// ---- GlobalTextList.TcGTLO
TEXTLIST GlobalTextList
  4330 = '\tPCW behavior Condition  (Suggestion from Intel)\n\tPCW SUPPLY THERMOCOUPLE LH\xa0 > 14°C, Warning: “PCW supply high temp”, Action: Nil\n\t(Tester) Incoming pressure for 6bar LH <550 kPa , Warning: “6 bar OFA LH air pressure low”,\xa0 Action: Nil\n\t(AP) Incoming pressure for 9 bar\xa0 LH < 850kPa, Warning:\xa0 “9 bar OFA LH air pressure low”, Action: Nil\n\tPCW Return Temperature – PCW Supply Temperature > 10degC, Warning: “Excessive heat load into PCW”, Action = Nil\n\tT-BOT Dew Point - PCW Supply Temperature > -2degC, Warning : “Dew point – PCW temperature above control limit, condensation warning.”, Action = Nil\n\tT-BOT Dew Point - PCW Supply Temperature > 0degC, Alarm: “Dew point – PCW temperature above critical control limit, condensation alarm.”, Action = Shut off PCW Supply and Return\n\tIf Either One of the Leak Sensor is Trigger, Alarm: “System PCW Leakage .”, Action = Shut off PCW Supply and Return.\n\t'
  1821 = '\tPCW behavior Condition  (Suggestion from Intel)\n\tPCW SUPPLY THERMOCOUPLE \xa0 > 14°C, Warning: “PCW supply high temp”, Action: Nil\n\t(Tester) Incoming pressure for 6bar  <550 kPa , Warning: “6 bar OFA LH air pressure low”,\xa0 Action: Nil\n\t(AP) Incoming pressure for 9 bar\xa0    < 850kPa, Warning:\xa0 “9 bar OFA LH air pressure low”, Action: Nil\n\tPCW Return Temperature – PCW Supply Temperature > 10degC, Warning: “Excessive heat load into PCW”, Action = Nil\n\tDew Point - PCW Supply Temperature > -2degC, Warning : “Dew point – PCW temperature above control limit, condensation warning.”, Action = Nil\n\tDew Point - PCW Supply Temperature > 0degC, Alarm: “Dew point – PCW temperature above critical control limit, condensation alarm.”, Action = Shut off PCW Supply and Return\n\tIf Either One of the Leak Sensor is Trigger, Alarm: “System PCW Leakage .”, Action = Shut off PCW Supply and Return.\n\t'
  3264 = '\tPCW behavior Condition  (Suggestion from Intel)\n\tPCW SUPPLY THERMOCOUPLE \xa0 > 14°C, Warning: “PCW supply high temp”, Action: Nil\n\t(Tester) Incoming pressure for 6bar  <550 kPa , Warning: “6 bar OFA LH air pressure low”,\xa0 Action: Nil\n\t(AP) Incoming pressure for 9 bar\xa0    < 850kPa, Warning:\xa0 “9 bar OFA LH air pressure low”, Action: Nil\n\tPCW Return Temperature – PCW Supply Temperature > 10degC, Warning: “Excessive heat load into PCW”, Action = Nil\n\tT-BOT Dew Point - PCW Supply Temperature > -2degC, Warning : “Dew point – PCW temperature above control limit, condensation warning.”, Action = Nil\n\tT-BOT Dew Point - PCW Supply Temperature > 0degC, Alarm: “Dew point – PCW temperature above critical control limit, condensation alarm.”, Action = Shut off PCW Supply and Return\n\tIf Either One of the Leak Sensor is Trigger, Alarm: “System PCW Leakage .”, Action = Shut off PCW Supply and Return.\n\t'
  571 = ' : '
  2622 = ' : AP Power Signal is not detected    '
  2268 = ' : AP Present Signal is not detected  '
  613 = ' : AP Ready Signal is not detected  '
  2271 = ' : APDeactuatedHwr Signal is not detected   '
  2182 = ' : APDeactuatedPLC Signal is not detected '
  2896 = ' : Cell Door Closed  Signal is not detected'
  3152 = ' : Cell Door Locked Signal is not detected'
  1060 = ' : Cell Fluid Leakage1 Signal is detected   '
  1608 = ' : Cell Fluid Leakage2  Signal is detecte'
  881 = ' : Cell Ground Fault Signal is detected     '
  4213 = ' : Debug Station Facility Ac Power OFF'
  3618 = ' : Debug Station Facility Ac Power OFF Detected'
  4041 = ' : DS cell fluid leakage 1 Signal is Detected'
  3638 = ' : DS cell fluid leakage 2 signal is detected'
  5457 = ' : e6BarLowOFAAirPressureAlarm'
  634 = ' : e6BarLowOFAAirPressureWarning'
  2402 = ' : e9BarLowOFAAirPressureWarning '
  3302 = ' : eCondensationWarning'
  639 = ' : eCriticalCondensationAlarm'
  244 = ' : eExcessiveHeatLoadIntoPCWWarning  '
  2432 = ' : ePCWSupplyHighTempWarning'
  6407 = ' : eSystemPCWLeakage2Alarm'
  1774 = ' : eSystemPCWLeakageAlarm'
  959 = ' : eSystemPCWReturnLeakageAlarm'
  3498 = ' : eSystemPCWSupplyLeakageAlarm'
  1221 = ' : Front Side Door Lock Signal is not Detected'
  3416 = ' : ipTCDrawerCylDown signal not detected'
  3147 = ' : ipTCDrawerCylExtendRS Signal not detected'
  1457 = ' : ipTCDrawerCylExtendRS signal not detected'
  3399 = ' : ipTCDrawerCylExtendRSError'
  1978 = ' : ipTCDrawerCylRetractRS signal not detected'
  7 = ' : ipTCDrawerCylRetractRSError'
  2361 = ' : ipTCDrawerCylUp signal not detected'
  137 = ' : nnnnn'
  1011 = ' : TBOT ANTI-COLLISION TRIGGERED SIGNAL'
  4581 = ' : TBot EAP AC Power OFF Detected'
  618 = ' : TBotEAPACPowerOFFDetected'
  2835 = ' : Tester Latches Closed  Signal is not detected '
  3173 = ' : Tester Present Signal is not detected  '
  2325 = ' : Tester Ready Signal is not detected  '
  700 = ' : TesterPower On  Signal is not detected '
  1694 = ' : TIU DOWN SOLENOID'
  957 = ' : TIU DOWN Solenoid Valve'
  4475 = ' : TIU EXTEND REED SWITCH'
  3125 = ' : TIU EXTEND SOLENOID'
  1932 = ' : TIU EXTEND Solenoid Valve'
  3331 = ' : TIU NOT SAFE TO MOVE'
  2540 = ' : TIU NOT SAFE TO MOVE (True: Not Safe, False Safe)'
  3756 = ' : TIU NOT SAFE TO MOVE (True:Not Safe,False: Safe)'
  3605 = ' : TIU NOT SAFETOMOVE (True:Not Safe,False: Safe)'
  1787 = ' : TIU Present Signal is not detected   '
  1466 = ' : TIU RETRACT REED SWITCH'
  1952 = ' : TIU RETRACT SOLENOID'
  2863 = ' : TIU RETRACT Solenoid Valve'
  4 = ' : TIU UP SOLENOID'
  1350 = ' : TIU UP Solenoid Valve'
  1123 = ' :(----------------------------------------------------------)'
  630 = ' :(--------------------------------------------------------------)'
  1673 = ' :(--------------------------------------------------------------------------------)'
  98 = ' :AP is not in UP Position'
  369 = ' :Both TIU Extern & Retract  Signal  are Detected'
  644 = ' :Both TIU Up & Down  Signal  are Detected'
  752 = ' :Door Close Signal is not Detected'
  2348 = ' :Door Lock Signal is not Detected'
  895 = ' :DrawerDownError'
  1112 = ' :DrawerExtendError'
  2406 = ' :DrawerRetractError'
  1818 = ' :DrawerUpError'
  4103 = ' :ipTCDrawerCylExtendRSError'
  1922 = ' :TBot EAP AntiCollision Triggered'
  4187 = ' :TBot EAP Not Safe To Move Error'
  2535 = ' :TBot EAPNotSofeToMoveError'
  2562 = ' :TBot Side Door Close Signal is not Detected'
  1220 = ' :TBot Side Door Lock Signal is not Detected'
  1668 = ' :TCC Session Active'
  4906 = '%3f'
  6313 = '%4.2'
  6022 = '%4.2f'
  1391 = '%5.0f'
  6312 = '%5.2'
  1806 = '%5.2f'
  2996 = '%6.3f'
  313 = '%d'
  5400 = '%D'
  311 = '%f'
  991 = '%i'
  4616 = '%s'
  3443 = '%t'
  3829 = "'C"
  1185 = '(----------------------------------------------------------------------------------)'
  632 = '(AP) OFA 10 bar Leak Flow'
  1515 = '(AP) OFA Pressure 10 bar'
  22 = '(Tester) OFA 6 bar Leak Flow'
  3541 = '(Tester) OFA Pressure 6 bar'
  4601 = '---------'
  234 = '01)Column Leakage'
  826 = '01)Col_Leakage'
  710 = '01)_AP_PresentSensor'
  3291 = '01)_AP_PresentSensor*'
  322 = '01)_Column Leakage'
  151 = '01)_ColumnLeakage'
  393 = '01)_Col_Leakage'
  427 = '02)_AllDrawerRetractedInCell'
  348 = '02)_All_Dwr_Ret'
  683 = '02)_AP_PowerOn'
  5106 = '02)_AP_PowerOn*'
  303 = '03)ColumnGround'
  976 = '03)_AP_Ready'
  75 = '03)_ColumnGround'
  941 = '03)_Col_Grd_Falt'
  1133 = '03)_Col_Grund_Falt'
  43 = '04)_AP_DeactuatedPLC'
  1100 = '04)_AP_DeactuatedPLC`*`'
  785 = '05)_AP_DeactuatedHwr'
  5223 = '05)_AP_DeactuatedHwr`*`'
  977 = '06)_CellFluidLeakage1'
  988 = '07)_CellFluidLeakage2'
  877 = '08)_CellGroundFault'
  421 = '09)_TesterPresent'
  2063 = '09)_TesterPresent*'
  2493 = '09)_TesterPresent**'
  1062 = '1'
  460 = "1'AP_PresentSenser"
  321 = '1)  AP_PresentSenser'
  671 = '1) AP_PresentSenser'
  566 = '1)_AP_PresentSensor'
  745 = '1)_Col_Leakage'
  537 = '1-AP_PresentSenser'
  2484 = '1. opDBStnMainPCWSupply'
  433 = '10)_TesterPowerOn'
  607 = '10)_TesterPowerOn*'
  729 = '10)_TesterPowerOn**'
  131 = '11)_TesterReady   '
  621 = '12)_TCCellDoorClosed\t'
  278 = '13)_TesterLatchesClosed'
  920 = '13)_TesterLatchesClosed**'
  117 = '14)_TIUPresent\t'
  577 = '2) AP_PowerOn'
  756 = '2)AP_PowerOn'
  129 = '2)_All_Dwr_Ret'
  628 = '2)_AP_PowerOn'
  1565 = '2. opDBStnPCWSupplyPurge'
  1692 = '21'
  2299 = '240 Power and PCW'
  4252 = '240v AP Power'
  5206 = '240v AP Power Feedback'
  2620 = '240v AP Power Feedback (Input)'
  4573 = '240v AP Power Feedback(Input)'
  2171 = '240v AP Power(Output)'
  4256 = '240v DPS/Tester Power'
  3856 = '240v Tester Power Feedback(Input)'
  1480 = '240v Tester Power(Output)'
  2285 = '240vTester Power(Output)'
  3074 = '240vTesterPower(Output)'
  846 = '3) AP_Ready'
  370 = '3)AP_Ready'
  145 = '3)_AP_Ready'
  1595 = '3)_Col_Grd'
  705 = '3)_Col_Grd_Falt'
  6218 = '3. opDBStnMainPCWReturn'
  84 = '4) AP_DeactuatedPLC'
  534 = '4)AP_DeactuatedPLC'
  965 = '4)_AP_DeactuatedPLC'
  1662 = '4. opDBStnPCWAWN'
  503 = '5) AP_DeactuatedHwr'
  559 = '5)AP_DeactuatedHwr'
  85 = '5)_AP_DeactuatedHwr'
  6470 = '5. opDBStnSupplyAirPurge'
  104 = '6)_CellFluidLeakage1'
  2776 = '6. opDBStnLeakFlowPCWValve'
  144 = '7)_CellFluidLeakage2'
  2027 = '7. opDBStnLowFlowPCWValve'
  51 = '8)_CellGroundFault'
  139 = '9)_TesterPresent'
  1420 = ': ColumnAlarmBit1'
  175 = ': ColumnAlarmBit2'
  658 = ': ColumnAlarmBit3'
  2042 = ': e6BarLowOFAAirPressureAlarm'
  5458 = ': ipTCDrawerCylRetractRSError'
  3543 = ': TBOT ANTI-COLLISION TRIGGERED SIGNAL'
  2700 = ': TBOT ANTI-COLLISION TRIGGERED SOGNAL'
  2570 = ': TIU EXTEND REED SWITCH'
  2097 = ': TIU NOT SAFE TO MOVE'
  3354 = ': TIU RETRACT REED SWITCH'
  2180 = ':AP is not in UP Position'
  4324 = ':ipTCDrawerCylRetractRSError'
  1467 = 'A'
  950 = 'AAAAAAAAAAA'
  3702 = 'Abort'
  2141 = 'Abort Running Timer'
  4237 = 'Abort Timer'
  5258 = 'Abort Timer (delay time)'
  312 = 'Actual Position'
  72 = 'Advanced'
  3639 = 'AH Alarm'
  3595 = 'AH Enable'
  4624 = 'AH SP'
  3633 = 'AHH Alarm'
  3579 = 'AHH Enable'
  3584 = 'AHH SP'
  2847 = 'Air Pressure Low'
  343 = 'Air Pressure Low ()'
  4556 = 'Air Pressure Low (Pressure is Less Than 550kpa)'
  2694 = 'Air Pressure Low (Pressure is less than 550kpa)'
  1084 = 'Air Pressure Low (Pressure is less than 850kPa)'
  3644 = 'AL Alarm'
  3600 = 'AL Enable'
  4631 = 'AL SP'
  5380 = 'Alar Auto Clearm'
  265 = 'Alarm'
  1301 = 'Alarm (Auto Clear)'
  1858 = 'Alarm Auto Clear'
  2577 = 'ALARM ID BIT STATUS'
  186 = 'ALARM ID BITS'
  690 = 'Alarm Reset'
  1223 = 'Alarm Running Timer'
  2152 = 'Alarm RunningTimer'
  2258 = 'Alarm Set PointWarning SetPoint'
  1212 = 'Alarm SetPoint'
  3433 = 'Alarm Timer'
  1638 = 'Alarm Timer (Second)'
  301 = 'Alarn Reset'
  3650 = 'ALL Alarm'
  3606 = 'ALL Enable'
  4638 = 'ALL SP'
  4995 = 'AllTCDrawer is not inside Cell'
  504 = 'AllTCDrawer_Not_In_Cell'
  5491 = 'AP 240Pwr Check Delay'
  1613 = 'AP Heater'
  1652 = 'AP HEATER_CURRENT'
  276 = 'AP is not in UP Position'
  5071 = 'AP Safe to Engage'
  2704 = 'AP240PwrCheck Delay(ms)'
  191 = 'AP240PwrCheckDelay(ms)'
  3283 = 'APReadyCheckDelay(ms)'
  81 = 'Auto'
  76 = 'Auto Input'
  624 = 'Auto Mode'
  469 = 'AutoRsetEvntTrigger'
  867 = 'BackDoorSimulationMode'
  1657 = 'Bar'
  633 = 'bar'
  252 = 'BH_HEATER_CURRENT_1'
  255 = 'BH_HEATER_CURRENT_2'
  254 = 'BH_HEATER_CURRENT_3'
  256 = 'BH_HEATER_CURRENT_4'
  1414 = 'BH_RTD_1'
  249 = 'BH_RTD_2'
  5795 = 'Btn No'
  1042 = 'Btn VIO Sim Override'
  6219 = 'Button'
  787 = 'Button: '
  1293 = 'ButtonModeConditionSimulation'
  1188 = 'ButtonModeConditionSimulation[iHMICbLevelSelection,iHMIBtnType]'
  535 = 'ButtonModeConditionSimulation[iHMICbLevelSelection,]'
  2089 = 'Cell Outputs :'
  1379 = 'Cell PCW'
  4038 = 'Cell Stack'
  2301 = 'CELL STACK'
  199 = 'Checkbox'
  2185 = 'Co'
  5100 = 'Col GroundFault'
  353 = 'COLUMN'
  2401 = 'Column'
  2816 = 'Column (AP) OFA Pressure 10 bar'
  329 = 'Column (Tester) OFA Pressure 6 bar'
  1708 = 'COLUMN ALARM ID BIT STATUS'
  4257 = 'COLUMN ALARM STATUS'
  2378 = 'Column Dew Point Sensor'
  3243 = 'Column Diagnostic Status'
  913 = 'Column Inputs :'
  90 = 'Column IO Diagnostic Mode'
  731 = 'Column Outputs :'
  2914 = 'Column PCW Leakage'
  3578 = 'Column PCW Regular Flow'
  2013 = 'Column PCW Return Pressure'
  2795 = 'Column PCW Return Temperature'
  2397 = 'Column PCW Supply Pressure'
  4011 = 'Column PCW Supply Temperature'
  1568 = 'Column Temperature'
  5977 = 'ColumnPCWLeakage2EAP'
  4652 = 'ColumnPCWLeakageEAP'
  2796 = 'ColumnPCWReturnLeakageEAP'
  760 = 'ColumnPCWSupplyLeakageEAP'
  5227 = 'Column_PCWLeakage'
  983 = 'Col_GroundFault'
  733 = 'Commands:'
  70 = 'Control'
  3437 = 'Current Value'
  272 = 'Cycle Running'
  4645 = 'DB'
  4543 = 'DBColumnPCWLeakage2EAP'
  3649 = 'DBColumnPCWLeakageEAP'
  4640 = 'DBColumnPCWReturnLeakageEAP'
  2584 = 'DBColumnPCWSupplyLeakageEAP'
  101 = 'DBColumnShutOffACPowerEAP'
  3120 = 'Dbug Station PCW Low Flow'
  270 = 'De Air Valve'
  1451 = 'De Pressure (Psi):'
  1001 = 'De Pressure Preset (Psi):'
  1464 = 'De Pressure Sen (Psi):'
  1689 = 'DE Stepping'
  4420 = 'DEBUG COLUMN ALARM ID BIT STATUS'
  3964 = 'DEBUG COLUMN ALARM STATUS'
  3330 = 'Debug Column Diagnostic Status'
  91 = 'Debug Column EAP Signals :'
  1164 = 'Debug Station'
  5185 = 'DEBUG STATION'
  2775 = 'Debug Station (AP) OFA 10 bar Leak Flow'
  1849 = 'Debug Station (Tester) OFA 6 bar Leak Flow'
  1416 = 'Debug Station Diagnostic Status'
  2458 = 'DEBUG STATION INPUTS'
  889 = 'DEBUG STATION IPC INPUTS'
  3105 = 'DEBUG STATION IPC OUTPUT'
  1865 = 'DEBUG STATION OUTPUT'
  271 = 'Debug Station PCW Leak Flow'
  488 = 'DeReg Pressure (Psi):'
  373 = 'DESolValve'
  541 = 'Development Purpose only'
  2911 = 'Dew Point '
  1678 = 'Dew Point - PCW Supply Temperature > -2degC, Warning :\nDew point – PCW temperature is above control limit, condensation warning'
  3845 = 'Dew Point - PCW Supply Temperature > -2degC, Warning : “Dew point – PCW temperature above control limit, condensation warning.”, Action = Nil'
  2334 = 'Dew Point - PCW Supply Temperature > 0degC, \nDew point – PCW temperature above critical control limit, condensation alarm\n'
  2414 = 'Dew Point - PCW Supply Temperature > 0degC, Alarm:\nDew point – PCW temperature above critical control limit, condensation alarm\n'
  4897 = 'Dew Point Alarm'
  3419 = 'Dew Point Dew Point '
  3035 = 'Dew Point Temperature'
  2356 = 'Dew Point Warning'
  1545 = 'Done Requested Action'
  1472 = 'Drawer In Request'
  1251 = 'Drawer Out Request'
  562 = 'Drawer Teaching Mode'
  1994 = 'DS_Facility_eapShutOffAllACPower'
  2386 = 'e6BarLowOFAAirPressureAlarm'
  398 = 'EAP SAFTY SIGNAL STATUS'
  1205 = 'EAP SAFTY SIGNAL STATUSSTATUS'
  2987 = 'EAP SIGNAL STATUS'
  3895 = 'eapShutOffAllACPower'
  948 = 'Enable'
  2173 = 'Enable Man: Stepping'
  1387 = 'Enable Man:Stepping'
  823 = 'Enable Manual Stepping Option'
  1120 = 'Enable Simulation'
  3674 = 'Enable/ Disable Status'
  1317 = 'EndPressure'
  2517 = 'EPT : '
  3022 = 'EPT States'
  314 = 'Error Code'
  4201 = 'Error Status: [ 0: No Error ]'
  1271 = 'Error Status: [0: No Error'
  2810 = 'ew Point Dew Point '
  83 = 'Extend'
  88 = 'Extended'
  2945 = 'F'
  2527 = 'Facility Alarm (Dew point & OFA6Bar)'
  3229 = 'Facility Alarm (Dew point & OFA6Bar) '
  4331 = 'Facility Alarm Set Default Timer and Point Value(Dew point & OFA6Bar) '
  4547 = 'Facility Alarm Set point and Timer'
  78 = 'Failed'
  80 = 'Failed to extend'
  79 = 'Failed to retract'
  1675 = 'For  Development And '
  4075 = 'Green: Enable , Gray: Disable'
  448 = 'Green:Enable , Gray: Disable'
  873 = 'GroupBox'
  3617 = 'Healthy'
  771 = 'Heater'
  1455 = 'HEATER_CURRENT_1'
  703 = 'HEATER_CURRENT_1:'
  1958 = 'HEATER_CURRENT_2'
  1131 = 'HEATER_CURRENT_3'
  500 = 'HEATER_CURRENT_4'
  1357 = 'Individual Alarm ID'
  1274 = 'Individual Alarm ID:'
  759 = 'Init All Level'
  3193 = 'INPUT'
  263 = 'Inputs :'
  636 = 'IO Diagnostic Mode'
  218 = 'ipAllTCDrawerRetractedinCell'
  734 = 'ipAPDeactuatedHwr'
  56 = 'ipAPDeactuatedPLC'
  715 = 'ipAPPowerOn'
  297 = 'ipAPPresentSensor'
  1003 = 'ipAPReady'
  409 = 'ipCellFluidLeakage1'
  994 = 'ipCellFluidLeakage2'
  611 = 'ipCellGroundFault'
  1030 = 'ipColumnFluid_PCW_Leakage'
  3804 = 'ipDBColumnPCWLeakage'
  1434 = 'ipDBColumnPCWLeakage2'
  777 = 'ipDBColumnPCWLeakageEAP'
  2983 = 'ipDBColumnPCWReturnLeakage'
  1794 = 'ipDBColumnPCWReturnLeakageEAP'
  631 = 'ipDBColumnPCWSupplyLeakage'
  3362 = 'ipDBColumnPCWSupplyLeakageEAP'
  2784 = 'ipDBStnAPDeactuatedHwr'
  1899 = 'ipDBStnAPDeactuatedPLC'
  1677 = 'ipDBStnAPPowerOn'
  1898 = 'ipDBStnAPPresentSensor'
  1372 = 'ipDBStnAPReady'
  2044 = 'ipDBStnCellFluidLeakage1'
  4211 = 'ipDBStnCellFluidLeakage2'
  2457 = 'ipDBStnCellGroundFault'
  1683 = 'ipDBStnPurgeButton'
  699 = 'ipDrawerMaintenanceModeBtn'
  6047 = 'ipFrontDoorClosed01'
  4595 = 'ipFrontDoorClosed02'
  3678 = 'ipFrontDoorLocked01'
  3016 = 'ipFrontDoorLocked02'
  502 = 'ipSpare_1'
  5492 = 'ipSpare_10'
  2251 = 'ipSpare_2'
  3485 = 'ipSpare_3'
  3951 = 'ipSpare_4'
  4430 = 'ipSpare_9'
  926 = 'ipSystemColumnGroundFault'
  5439 = 'ipTbotDoorClosedSignal'
  3073 = 'ipTbotDoorClosedSignal not Detected'
  934 = 'ipTCCellAbortFlowBtn'
  161 = 'ipTCCellDoorClosed'
  1318 = 'ipTCCellDoorLocked'
  42 = 'ipTCCellDoorOpenCloseStatus'
  743 = 'ipTCCellDoorOpenReqBtn'
  4199 = 'ipTCCellFrontDoorOpenCloseStatus01'
  3873 = 'ipTCCellTbotSideDoorLocked01'
  2955 = 'ipTCCellTbotSideDoorLocked02'
  2696 = 'ipTCCellTbotSideDoorOpenCloseStatus01'
  2935 = 'ipTCCellTbotSideDoorOpenCloseStatus02'
  844 = 'ipTCDrawerCylDownRS'
  300 = 'ipTCDrawerCylExtendRS'
  1121 = 'ipTCDrawerCylRetractRS'
  346 = 'ipTCDrawerCylUpRS'
  660 = 'ipTesterLatchesClosed'
  600 = 'ipTesterPowerOn'
  228 = 'ipTesterPresent'
  647 = 'ipTesterReady'
  1132 = 'ipTIUPresent'
  617 = 'KPa'
  1810 = 'l/min'
  821 = 'L/min'
  224 = 'Label'
  1934 = 'Label:'
  341 = 'larm Set PointWarning SetPoint'
  69 = 'Leve l1'
  225 = 'Level'
  2252 = 'Level 1  : '
  5610 = 'Level 1 : '
  865 = 'Level 1 IO Diagnostic Mode'
  5436 = 'Level 2 : '
  374 = 'Level 3 : '
  6242 = 'Level 4 : '
  7414 = 'Level 5 : '
  6758 = 'Level 6 : '
  1000 = 'Level1 Inputs :'
  334 = 'Level1 Outputs :'
  405 = 'Level:'
  456 = 'Level[1]'
  540 = 'Level[1]:'
  501 = 'Level[2]'
  62 = 'Level[2]:'
  1891 = 'Level[3]'
  260 = 'Level[3]:'
  4747 = 'Level[4]'
  902 = 'Level[4]:'
  4654 = 'Level[5]'
  622 = 'Level[5]:'
  3942 = 'Level[6]'
  267 = 'Level[6]:'
  5482 = 'LowLow Set Point'
  623 = 'Main Air Valve'
  253 = 'Manual button Number'
  4489 = 'Manual Button Number'
  1985 = 'Manual Command Simulation From PLC'
  732 = 'Manual Command Test'
  625 = 'Manual Mode'
  1640 = 'Manual Solenoid Number'
  73 = 'Message'
  46 = 'mL/min'
  2246 = 'ml/min'
  3307 = 'Mod Enable Status'
  4077 = 'ModEnable Status'
  1832 = 'Module Enable Status'
  307 = 'MoveAbs'
  308 = 'MoveRel'
  1532 = 'Mpa'
  487 = 'No Of Cycle'
  1300 = 'NoStep'
  4859 = 'Note: This EAP is to shut off debug cell stack AC Power'
  5953 = 'Note: This is to shut off debug cell stack AC Power'
  1841 = 'OFA 10 bar Leak Flow'
  1801 = 'OFA 6 bar Leak Flow'
  1712 = 'OFA Pressure 10 bar'
  3060 = 'OFA Pressure 6 bar'
  342 = 'OFA6Bar'
  5648 = 'OFA6Bar Alarm'
  4462 = 'OFA6Bar Pressure'
  3791 = 'OFA6Bar Warning'
  4012 = 'OFA6BarPresessure'
  3379 = 'OFA6BarPresuure '
  2385 = 'Only For  Development'
  2157 = 'Only For  Development And '
  1313 = 'Only For Development'
  4886 = 'Only For Development &'
  868 = 'opACSSR1'
  1403 = 'opACSSR2'
  1795 = 'opACSSR3'
  1963 = 'opACSSR4'
  325 = 'opAlarmLED'
  21 = 'opAP240ACPwrEnable'
  8 = 'opAPAirSupplySol'
  4382 = 'opAPSafeToEngage'
  431 = 'opAPSafeToMoveSignal'
  744 = 'opAPTBD'
  5 = 'opAPTCCReset'
  50 = 'opAPTIUSktAir'
  447 = 'opAPTIUSktCoolingAir1'
  1423 = 'opAPTIUSktCoolingAir2'
  1476 = 'opAP_DIO_1'
  1905 = 'opAP_DIO_2'
  3970 = 'opAP_DIO_3'
  582 = 'opASCOValve_1 '
  1637 = 'opASCOValve_2'
  860 = 'opCell24VPowerEnable'
  1041 = 'opCellDoorClosed'
  4015 = 'opCellDoorLock'
  1225 = 'opCellDrawerCylDown'
  643 = 'opCellDrawerCylExtend'
  1104 = 'opCellDrawerCylRetract'
  248 = 'opCellDrawerCylUp'
  1037 = 'opCellLTIMValve'
  118 = 'opCellPCWValve'
  2608 = 'opCellTBotSideDoorClosed1'
  468 = 'opCellTBotSideDoorClosed1(DC)'
  2421 = 'opCellTBotSideDoorClosed1(DC),'
  3551 = 'opCellTBotSideDoorClosed2(DC)'
  1228 = 'opD'
  1255 = 'opDBColumnAPAirSol'
  3078 = 'opDBColumnHotAirExhaustFan'
  3176 = 'opDBColumnPCWValve'
  583 = 'opDBColumnTstAirSol'
  1125 = 'opDBStn24VPowerEnable  '
  2059 = 'opDBStnAlarmLED'
  1720 = 'opDBStnAP240ACPwrEnable'
  6059 = 'opDBStnAP30ACPwrEnable'
  689 = 'opDBStnAPSafeToMoveSignal    '
  1625 = 'opDBStnAPTCCReset  '
  4163 = 'opDBStnBypassAPAirSupplySol'
  1701 = 'opDBStnBypassAPAirSupplySol '
  366 = 'opDBStnLeakFlowPCWValve'
  5507 = 'opDBStnLeakFlowPCWValve*'
  3010 = 'opDBStnLowFlowPCWValve   '
  3011 = 'opDBStnLowFlowPCWValve* '
  3995 = 'opDBStnMainPCWReturn'
  2023 = 'opDBStnMainPCWSupply'
  1327 = 'opDBStnMainPCWValve'
  2648 = 'opDBStnPCWAWN'
  3509 = 'opDBStnPCWFlowBypassValve'
  2747 = 'opDBStnPCWFlowBypassValve*'
  924 = 'opDBStnPCWSupplyPurge'
  588 = 'opDBStnPCWValve'
  1291 = 'opDBStnPCWValve                 '
  2699 = 'opDBStnPurgeLED'
  324 = 'opDoorOpenReqLED'
  1230 = 'opDrawerMaintenanceModeBtnLED'
  1081 = 'opFrontDoorLock (DC)'
  1695 = 'opFrontDoorLock1 (DC)'
  4695 = 'opFrontDoorLock2 (DC)'
  880 = 'opHotAirExhaustFan'
  1366 = 'opMainIncomingAirValve'
  590 = 'opPowerEnable'
  5110 = 'opSpare_1'
  5152 = 'opSpare_10'
  60 = 'opSpare_2'
  3076 = 'opSpare_3'
  169 = 'opSpare_9'
  1092 = 'opTCCellAbortFlowBtnLED'
  354 = 'opTesterDrawerAirSupplySol'
  1124 = 'opTst240VACPwrEnable'
  1539 = 'OUTPUT'
  264 = 'Outputs :'
  560 = 'Override By HMI'
  1055 = 'Override DebugColumn IO'
  2314 = 'Override DebugStation IO'
  2991 = 'Override IO'
  220 = 'Override TII Alm Enable By HMI'
  528 = 'Override TII Alm EnableBy HMI'
  522 = 'Override TII Sen Simulation By HMI'
  1498 = 'PCW Leak Flow'
  2318 = 'PCW Low Flow'
  1424 = 'PCW Regular Flow'
  465 = 'PCW Regular Flow Meter'
  945 = 'PCW Return Pressure'
  1174 = 'PCW Return Temperature'
  2380 = 'PCW Supply Pressure'
  1415 = 'PCW Supply Temperature'
  1134 = 'PLC IO Diagnostic Mode'
  2665 = 'PLC IO DiagnosticMode'
  4112 = 'Process State'
  4472 = 'Process States'
  52 = 'Production Mode'
  4008 = 'Production Mode: '
  3611 = 'PV'
  1775 = 'Regular Flow Meter'
  310 = 'Reset'
  550 = 'Reset All'
  143 = 'Reset All Alarm'
  911 = 'Reset All ID'
  391 = 'Reset All Reset All Alarm'
  1626 = 'Reset Stepping'
  1329 = 'Result'
  82 = 'Retract'
  87 = 'Retracted'
  1578 = 'RTD_1:'
  1214 = 'RTD_2'
  1463 = 'RTD_2:'
  987 = 'Save'
  6434 = 'sdsdsds'
  6062 = 'Sec'
  4062 = 'Second'
  4470 = 'Seconds'
  323 = 'SenL[1]'
  973 = 'SenL[1] Sim'
  123 = 'SenL[2]:'
  332 = 'Set'
  315 = 'Set Absolute Pos'
  316 = 'Set Absolute Speed'
  417 = 'Set No Of Cycle'
  317 = 'Set Rel Pos'
  318 = 'Set Rel Speed'
  3589 = 'Settings'
  3622 = 'Simulate'
  77 = 'Simulation'
  4852 = 'Simulation Mode'
  233 = 'SOFT EAP SIGNAL STATUS'
  2950 = 'SOFT SAFTY SIGNAL STATUS'
  1897 = 'Sorly  For  Development And '
  4398 = 'Sorly Development And Troubleshooting Purpose only'
  1105 = 'Sorly For Development And '
  268 = 'Spare'
  74 = 'Start'
  1311 = 'StartPressure'
  1305 = 'StartStepping'
  7134 = 'State Timer'
  3628 = 'Status'
  1322 = 'SteppingDelay'
  309 = 'Stop'
  720 = 'System Alarm'
  7074 = 'System Mode:'
  266 = 'System Ready'
  4689 = 'TC COLUMN ALARM STATUS'
  258 = 'TC1_INLET '
  259 = 'TC4_OUTLET'
  2762 = 'TCU '
  3428 = 'TCU Enable Status'
  269 = 'Te Air Valve'
  1005 = 'Te Pressure (Psi):'
  996 = 'Te Pressure Preset (Psi):'
  1456 = 'Te Pressure Sen (Psi):'
  1232 = 'TE Stepping'
  626 = 'Te Up Sensor'
  1450 = 'TE Up Sensor'
  1840 = 'TE/DE Input'
  345 = 'TE/DE Manual Stepping'
  1409 = 'TE/DE Output'
  629 = 'TEDE Output'
  614 = 'TeReg Pressure (Psi):'
  1166 = 'TESolValve'
  2541 = 'TessterEnable Status'
  425 = 'Test Command'
  1972 = 'Tester'
  1735 = 'TESTER '
  2201 = 'TESTER CELL'
  2997 = 'TESTER CELL  '
  1697 = 'TESTER CELL :'
  380 = 'TESTER CELL ::'
  250 = 'TH_HEATER_CURRENT_1'
  251 = 'TH_HEATER_CURRENT_2'
  1398 = 'TH_RTD_1:'
  1406 = 'TH_RTD_2'
  320 = 'TierII Alarm'
  4887 = 'TII'
  1490 = 'TII Alarm Enable Override'
  4170 = 'TII Enable Status'
  4356 = 'TII Enable/Disable Status'
  2282 = 'TII Sen: VIO Sim Override'
  3444 = 'TII Sen:VIO Sim Override'
  1418 = 'TII VIO Sim Override'
  5232 = 'TIISen:VIO Sim Override'
  2075 = 'TIISen:VIOSim Override'
  561 = 'TIIVIO Simulate Override'
  1438 = 'TIIVIO Simulation Override'
  86 = 'Travel time:'
  1191 = 'Troubleshooting Purpose only !'
  645 = 'Troubleshooting use !'
  946 = 'Troubleshooting use only !'
  843 = 'Tst 240Pwr Check Delay'
  3770 = 'Tst240PwrCheckDelay(ms)'
  3842 = 'TstReadyCheckDelay(ms)'
  319 = 'Up'
  5055 = 'Value to Write'
  4930 = 'Value To Write'
  595 = 'VIO Simulation Override'
  408 = 'VIO Status'
  1024 = 'Vir IO Simulation'
  1328 = 'Vir IO Simulation Override'
  71 = 'Warning'
  7498 = 'Warning Running Timer'
  6812 = 'Warning RunningTimer'
  5722 = 'Warning SetPoint'
  4110 = 'Warning SetPoint        <'
  2400 = 'Warning SetPoint    <'
  4641 = 'Warning Timer'
  330 = 'Warning Timer (second)'
  778 = 'Warning Tinmer'
  1848 = 'WaterValve'
  2341 = 'wewewwwewewDew Point '
  1362 = 'Write'
  4658 = 'wwewewDew Point '
  794 = 'zz'
  2132 = '[ 01 ]:'
  328 = '[ 02 ]:'
  949 = '[ 03 ]:'
  89 = '[ 04 ]:'
  1051 = '[ 05 ]:'
  2327 = '[ 06 ]:'
  35 = '[ 07 ]:'
  1326 = '[ 08 ]:'
  1095 = '[ 09 ]:'
  979 = '[ 10 ]:'
  2390 = '[ 11 ]:'
  969 = '[ 12 ]:'
  575 = '[ 13 ]:'
  274 = '[ 14 ]:'
  615 = '[ 15 ]:'
  2494 = '[ 16 ]:'
  1006 = '[ 17 ]:'
  168 = '[ 18 ]:'
  2717 = '[ 19 ]:'
  2826 = '[ 20 ]:'
  2437 = '[ 21 ]'
  1871 = '[ 21 ]:'
  326 = '[ 22 ]:'
  1649 = '[ 23 ]:'
  1936 = '[ 24 ]:'
  616 = '[ 240 Power and PCW: ]'
  1437 = '[ 24]:'
  1449 = '[ 25 ]:'
  2279 = '[ 26 ]:'
  2434 = '[ 27 ]:'
  1951 = '[ 28 ]:'
  1330 = '[ 29 ]:'
  327 = '[ 30 ]:'
  2518 = '[ 31 ]:'
  1653 = '[ 32 ]:'
  627 = '[ 33 ]:'
  1349 = '[ 34 ]:'
  638 = '[ 35 ]:'
  569 = '[ 36 ]:'
  816 = '[ 37 ]:'
  2486 = '[ 38 ]:'
  340 = '[ 39 ]:'
  2266 = '[ 40 ]:'
  1600 = '[ 41 ]:'
  2080 = '[ 41]:'
  1751 = '[ 42 ]:'
  358 = '[ 43 ]:'
  1056 = '[ 44 ]:'
  1511 = '[ 45 ]:'
  2429 = '[ 46 ]:'
  4935 = '[ 47 ]:'
  5024 = '[ 48 ]:'
  7540 = '[ 49 ]:'
  5360 = '[ 50 ]:'
  799 = '[ 51 ]:'
  5358 = '[ 52 ]:'
  5316 = '[ 53 ]:'
  7608 = '[ 54 ]:'
  6453 = '[ 55 ]:'
  1516 = '[ P1]:'
  1336 = '[ P2]:'
  3163 = '[ P3]:'
  3117 = '[ P4]:'
  2215 = '[ P5]:'
  2300 = '[ P6]:'
  3705 = '[ Pub1]:'
  1045 = '[ S1]:'
  3115 = '[ S2]:'
  1529 = '[ S3]:'
  3009 = '[ S4]:'
  1198 = '[ S5]:'
  1570 = '[ S6]:'
  1700 = '[21]'
  5455 = '°C'
END_TEXTLIST

// ---- GVLs/AlarmTxtList.TcTLO
TEXTLIST AlarmTxtList
  1 = "'AP_PresentSensor'"
  2 = "'AP_PowerOn'"
  3 = "'AP_Ready'"
  4 = "'AP_DeactuatedPLC' "
  5 = "'AP_DeactuatedHwr' "
  6 = "'CellFluidLeakage1' "
  7 = "'CellFluidLeakage2' "
  8 = "'CellGroundFault' "
  9 = "'TesterPresent' "
  10 = "'TesterPowerOn'"
  11 = "'TesterReady' "
  12 = "'TCCellDoorClosed'"
  13 = "'TesterLatchesClosed'"
  14 = "'TIUPresent'"
  15 = ''
  16 = ''
   = ''
END_TEXTLIST

// ---- GVLs/BDList.TcTLO
TEXTLIST BDList
  0 = 'Disable'
  1 = 'ForceOn'
  2 = 'ForceOff'
   = ''
END_TEXTLIST

// ---- GVLs/BtnTxtList.TcTLO
TEXTLIST BtnTxtList
  1 = '1. MaintenanceButton'
  2 = '2. AbortFlowButton'
  3 = '3. DoorUnlockButton'
  4 = 'emtpy'
  5 = '5. PurgeFlowbutton'
   = ''
END_TEXTLIST

// ---- GVLs/CmdTxtList.TcTLO
TEXTLIST CmdTxtList
  0 = 'INITIALISE'
  1 = 'AlarmReset'
  2 = 'ColumnAlarmReset'
  3 = 'TIUSlideIn'
  4 = 'TIUSlideOut'
  5 = 'TIUDrawerUp'
  6 = 'TIUDrawerDown'
  7 = 'TIUSlideOutRetry'
  8 = 'TIUSlideOutCancel'
  9 = 'DPSPowerON'
  10 = 'DPSPowerOFF'
  11 = 'DPSPowerAuto'
  12 = 'AP240ACPowerON'
  13 = 'AP240ACPowerOFF'
  14 = 'APAirValveON'
  15 = 'APAirValveOFF'
  16 = 'TstAirValveON'
  17 = 'TstAirValveOFF'
  18 = 'CellDoorOpen'
  19 = 'CellDoorClose'
  20 = 'CancelBuffer'
  21 = 'SetLEDON'
  22 = 'SetLEDOFF'
  23 = 'SetLEDBlink'
  24 = 'DCCellFrontDoorOpen'
  25 = 'DCCellFrontDoorClose'
  26 = 'TIUSocketAirOn_1'
  27 = 'TIUSocketAirOn_2'
  28 = 'TIUSocketAirOff_1'
  29 = 'TIUSocketAirOff_2'
  30 = 'EnableTester'
  31 = 'DisableTester'
  32 = 'EnableTCU'
  33 = 'DisableTCU'
  34 = 'EnableTII'
  35 = 'DisableTII'
  36 = 'SetTCUSafeState'
  37 = 'SetSolenoidValvesON'
  38 = 'SetSolenoidValvesOFF'
  39 = 'Secondary24VPowerON'
  40 = 'Secondary24VPowerOFF'
   = ''
END_TEXTLIST

// ---- GVLs/LevelTxtList.TcTLO
TEXTLIST LevelTxtList
  1 = 'level [1]'
  2 = 'level [2]'
  3 = 'level [3]'
  4 = 'level [4]'
  5 = 'level [5]'
  6 = 'level [6]'
   = ''
END_TEXTLIST

// ---- VISUs/HMI_Alarm.TcVIS
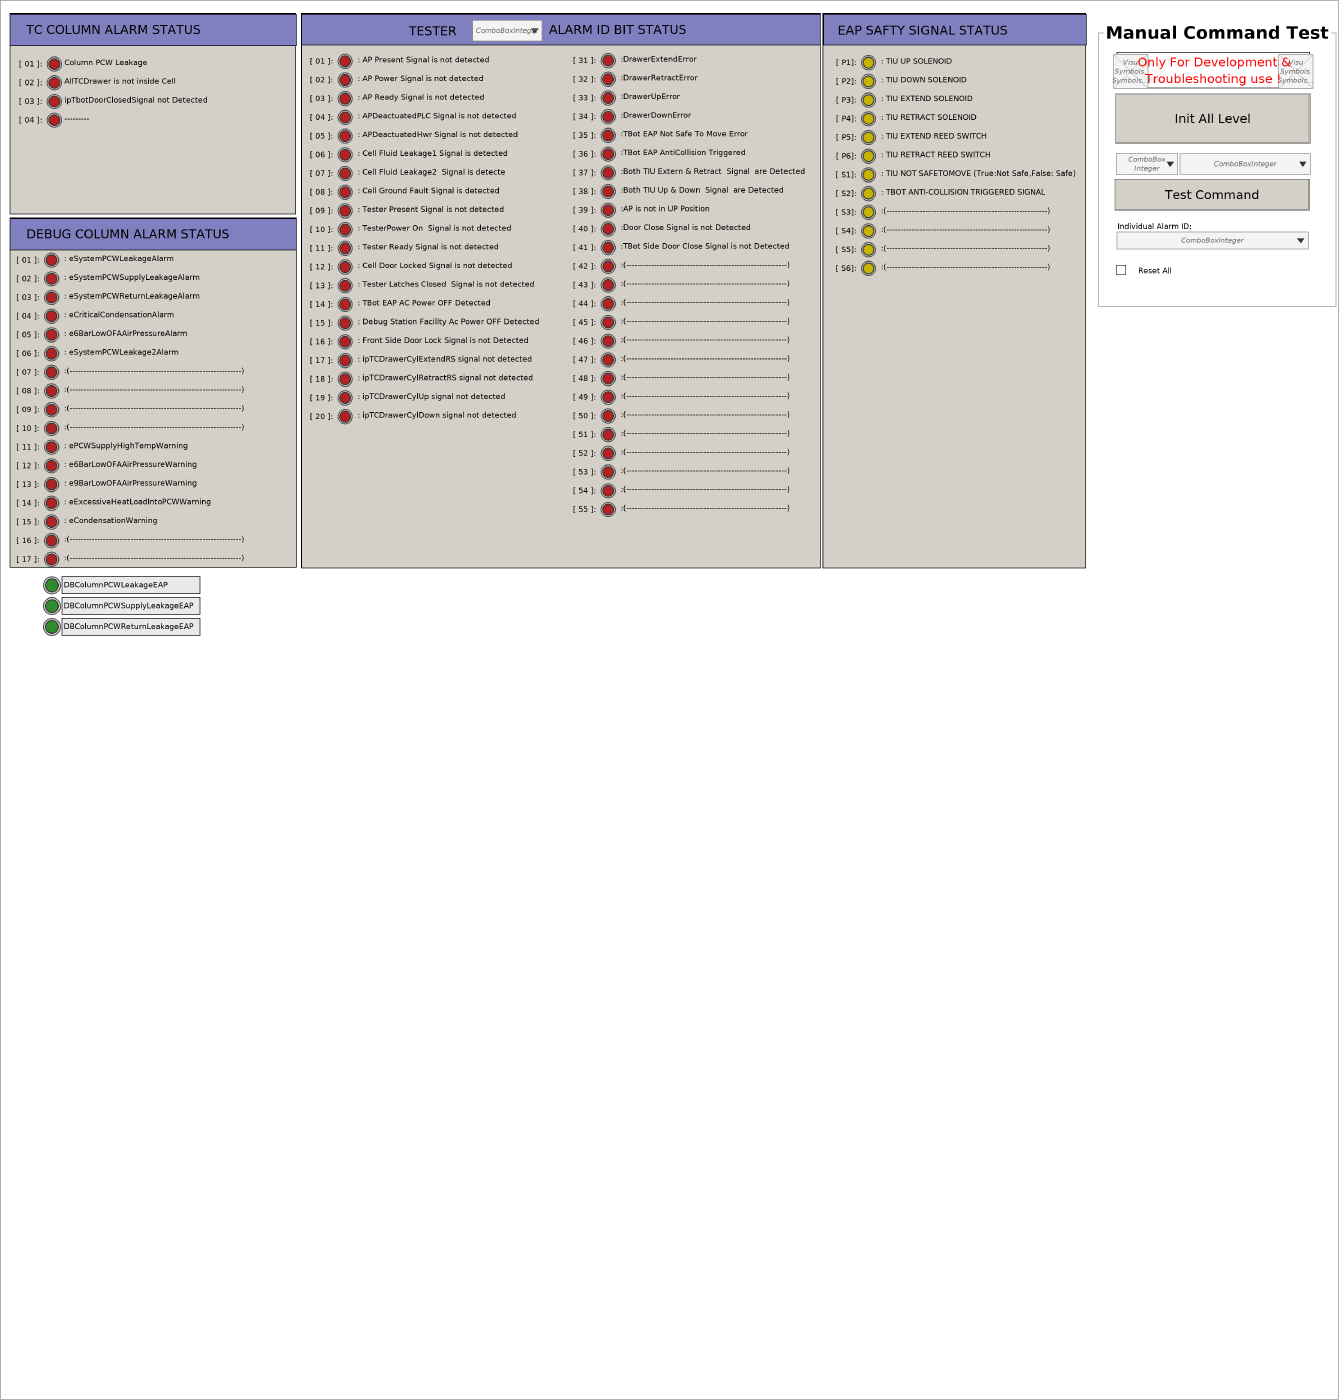
VISUALIZATION HMI_Alarm  // 1934x2021
    Rectangle (1188,19 380x801)
    Rectangle (1189,20 380x45)
    Rectangle (435,19 750x801)
    Rectangle (435,20 750x45)
    Rectangle (14,19 413x290)
    Rectangle (14,20 414x46)
    Lamp1 (866,75 25x25), variable: ALMTC.Level[iHMICbLevelSelection].AlarmID[31], style: Lamp-Lamp1-Red
    Label (824,75 40x25), "[ 31 ]:"
    Label (890,73 300x25), ":DrawerExtendError"
    ComboBoxInteger (682,29 101x30), variable: iHMICbLevelSelection, text list: 'LevelTxtList'
    Lamp1 (866,102 25x25), variable: ALMTC.Level[iHMICbLevelSelection].AlarmID[32], style: Lamp-Lamp1-Red
    Label (824,102 40x25), "[ 32 ]:"
    Label (890,100 300x25), ":DrawerRetractError"
    Lamp1 (866,129 25x25), variable: ALMTC.Level[iHMICbLevelSelection].AlarmID[33], style: Lamp-Lamp1-Red
    Label (824,129 40x25), "[ 33 ]:"
    Label (890,127 300x25), ":DrawerUpError"
    Lamp1 (866,156 25x25), variable: ALMTC.Level[iHMICbLevelSelection].AlarmID[34], style: Lamp-Lamp1-Red
    Label (824,156 40x25), "[ 34 ]:"
    Label (890,154 300x25), ":DrawerDownError"
    Lamp1 (866,183 25x25), variable: ALMTC.Level[iHMICbLevelSelection].AlarmID[35], style: Lamp-Lamp1-Red
    Label (824,183 40x25), "[ 35 ]:"
    Label (890,181 300x25), ":TBot EAP Not Safe To Move Error"
    Lamp1 (866,210 25x25), variable: ALMTC.Level[iHMICbLevelSelection].AlarmID[36], style: Lamp-Lamp1-Red
    Label (824,210 40x25), "[ 36 ]:"
    Label (890,208 300x25), ":TBot EAP AntiCollision Triggered"
    Lamp1 (866,237 25x25), variable: ALMTC.Level[iHMICbLevelSelection].AlarmID[37], style: Lamp-Lamp1-Red
    Label (824,237 40x25), "[ 37 ]:"
    Label (890,235 300x25), ":Both TIU Extern & Retract Signal are Detected"
    Lamp1 (866,264 25x25), variable: ALMTC.Level[iHMICbLevelSelection].AlarmID[38], style: Lamp-Lamp1-Red
    Label (824,264 40x25), "[ 38 ]:"
    Label (890,262 300x25), ":Both TIU Up & Down Signal are Detected"
    Lamp1 (866,291 25x25), variable: ALMTC.Level[iHMICbLevelSelection].AlarmID[39], style: Lamp-Lamp1-Red
    Label (824,291 40x25), "[ 39 ]:"
    Label (890,289 300x25), ":AP is not in UP Position"
    Lamp1 (866,318 25x25), variable: ALMTC.Level[iHMICbLevelSelection].AlarmID[40], style: Lamp-Lamp1-Red
    Label (824,318 40x25), "[ 40 ]:"
    Label (890,316 300x25), ":Door Close Signal is not Detected"
    Lamp1 (866,345 25x25), variable: ALMTC.Level[iHMICbLevelSelection].AlarmID[41], style: Lamp-Lamp1-Red
    Label (824,345 40x25), "[ 41 ]:"
    Label (890,343 300x25), ":TBot Side Door Close Signal is not Detected"
    Lamp1 (866,372 25x25), variable: ALMTC.Level[iHMICbLevelSelection].AlarmID[42], style: Lamp-Lamp1-Red
    Label (824,372 40x25), "[ 42 ]:"
    Label (890,370 300x25), ":(----------------------------------------------------------)"
    Lamp1 (866,399 25x25), variable: ALMTC.Level[iHMICbLevelSelection].AlarmID[43], style: Lamp-Lamp1-Red
    Label (824,399 40x25), "[ 43 ]:"
    Label (890,397 300x25), ":(----------------------------------------------------------)"
    Lamp1 (866,426 25x25), variable: ALMTC.Level[iHMICbLevelSelection].AlarmID[44], style: Lamp-Lamp1-Red
    Label (824,426 40x25), "[ 44 ]:"
    Label (890,424 300x25), ":(----------------------------------------------------------)"
    Lamp1 (866,453 25x25), variable: ALMTC.Level[iHMICbLevelSelection].AlarmID[45], style: Lamp-Lamp1-Red
    Label (824,453 40x25), "[ 45 ]:"
    Label (890,451 300x25), ":(----------------------------------------------------------)"
    Lamp1 (866,480 25x25), variable: ALMTC.Level[iHMICbLevelSelection].AlarmID[46], style: Lamp-Lamp1-Red
    Label (824,480 40x25), "[ 46 ]:"
    Label (890,478 300x25), ":(----------------------------------------------------------)"
    Lamp1 (866,507 25x25), variable: ALMTC.Level[iHMICbLevelSelection].AlarmID[47], style: Lamp-Lamp1-Red
    Label (824,507 40x25), "[ 47 ]:"
    Label (890,505 300x25), ":(----------------------------------------------------------)"
    Lamp1 (866,534 25x25), variable: ALMTC.Level[iHMICbLevelSelection].AlarmID[48], style: Lamp-Lamp1-Red
    Label (824,534 40x25), "[ 48 ]:"
    Label (890,532 300x25), ":(----------------------------------------------------------)"
    Lamp1 (866,561 25x25), variable: ALMTC.Level[iHMICbLevelSelection].AlarmID[49], style: Lamp-Lamp1-Red
    Label (824,561 40x25), "[ 49 ]:"
    Label (890,559 300x25), ":(----------------------------------------------------------)"
    Lamp1 (866,588 25x25), variable: ALMTC.Level[iHMICbLevelSelection].AlarmID[50], style: Lamp-Lamp1-Red
    Label (824,588 40x25), "[ 50 ]:"
    Label (890,586 300x25), ":(----------------------------------------------------------)"
    Lamp1 (866,615 25x25), variable: ALMTC.Level[iHMICbLevelSelection].AlarmID[50], style: Lamp-Lamp1-Red
    Label (824,615 40x25), "[ 51 ]:"
    Label (890,613 300x25), ":(----------------------------------------------------------)"
    Lamp1 (866,642 25x25), variable: ALMTC.Level[iHMICbLevelSelection].AlarmID[50], style: Lamp-Lamp1-Red
    Label (824,642 40x25), "[ 52 ]:"
    Label (890,640 300x25), ":(----------------------------------------------------------)"
    Lamp1 (866,669 25x25), variable: ALMTC.Level[iHMICbLevelSelection].AlarmID[50], style: Lamp-Lamp1-Red
    Label (824,669 40x25), "[ 53 ]:"
    Label (890,667 300x25), ":(----------------------------------------------------------)"
    Lamp1 (866,696 25x25), variable: ALMTC.Level[iHMICbLevelSelection].AlarmID[50], style: Lamp-Lamp1-Red
    Label (824,696 40x25), "[ 54 ]:"
    Label (890,694 300x25), ":(----------------------------------------------------------)"
    Lamp1 (866,723 25x25), variable: ALMTC.Level[iHMICbLevelSelection].AlarmID[50], style: Lamp-Lamp1-Red
    Label (824,723 40x25), "[ 55 ]:"
    Label (890,721 300x25), ":(----------------------------------------------------------)"
    Lamp1 (486,76 25x25), variable: ALMTC.Level[iHMICbLevelSelection].AlarmID[1], style: Lamp-Lamp1-Red
    Label (444,76 40x25), "[ 01 ]:"
    Label (510,74 300x25), ": AP Present Signal is not detected"
    Lamp1 (486,103 25x25), variable: ALMTC.Level[iHMICbLevelSelection].AlarmID[2], style: Lamp-Lamp1-Red
    Label (444,103 40x25), "[ 02 ]:"
    Label (510,101 300x25), ": AP Power Signal is not detected"
    Lamp1 (486,130 25x25), variable: ALMTC.Level[iHMICbLevelSelection].AlarmID[3], style: Lamp-Lamp1-Red
    Label (444,130 40x25), "[ 03 ]:"
    Label (510,128 300x25), ": AP Ready Signal is not detected"
    Lamp1 (486,157 25x25), variable: ALMTC.Level[iHMICbLevelSelection].AlarmID[4], style: Lamp-Lamp1-Red
    Label (444,157 40x25), "[ 04 ]:"
    Label (510,155 300x25), ": APDeactuatedPLC Signal is not detected"
    Lamp1 (486,184 25x25), variable: ALMTC.Level[iHMICbLevelSelection].AlarmID[5], style: Lamp-Lamp1-Red
    Label (444,184 40x25), "[ 05 ]:"
    Label (510,182 300x25), ": APDeactuatedHwr Signal is not detected"
    Lamp1 (486,211 25x25), variable: ALMTC.Level[iHMICbLevelSelection].AlarmID[6], style: Lamp-Lamp1-Red
    Label (444,211 40x25), "[ 06 ]:"
    Label (510,209 300x25), ": Cell Fluid Leakage1 Signal is detected"
    Lamp1 (486,238 25x25), variable: ALMTC.Level[iHMICbLevelSelection].AlarmID[7], style: Lamp-Lamp1-Red
    Label (444,238 40x25), "[ 07 ]:"
    Label (510,236 300x25), ": Cell Fluid Leakage2 Signal is detecte"
    Lamp1 (486,265 25x25), variable: ALMTC.Level[iHMICbLevelSelection].AlarmID[8], style: Lamp-Lamp1-Red
    Label (444,265 40x25), "[ 08 ]:"
    Label (510,263 300x25), ": Cell Ground Fault Signal is detected"
    Lamp1 (486,292 25x25), variable: ALMTC.Level[iHMICbLevelSelection].AlarmID[9], style: Lamp-Lamp1-Red
    Label (444,292 40x25), "[ 09 ]:"
    Label (510,290 300x25), ": Tester Present Signal is not detected"
    Lamp1 (486,319 25x25), variable: ALMTC.Level[iHMICbLevelSelection].AlarmID[10], style: Lamp-Lamp1-Red
    Label (444,319 40x25), "[ 10 ]:"
    Label (510,317 300x25), ": TesterPower On Signal is not detected"
    Lamp1 (486,346 25x25), variable: ALMTC.Level[iHMICbLevelSelection].AlarmID[11], style: Lamp-Lamp1-Red
    Label (444,346 40x25), "[ 11 ]:"
    Label (510,344 300x25), ": Tester Ready Signal is not detected"
    Lamp1 (486,373 25x25), variable: ALMTC.Level[iHMICbLevelSelection].AlarmID[12], style: Lamp-Lamp1-Red
    Label (444,373 40x25), "[ 12 ]:"
    Label (510,371 300x25), ": Cell Door Locked Signal is not detected"
    Lamp1 (486,400 25x25), variable: ALMTC.Level[iHMICbLevelSelection].AlarmID[13], style: Lamp-Lamp1-Red
    Label (444,400 40x25), "[ 13 ]:"
    Label (510,398 300x25), ": Tester Latches Closed Signal is not detected"
    Lamp1 (486,427 25x25), variable: ALMTC.Level[iHMICbLevelSelection].AlarmID[14], style: Lamp-Lamp1-Red
    Label (444,427 40x25), "[ 14 ]:"
    Label (510,425 300x25), ": TBot EAP AC Power OFF Detected"
    Lamp1 (486,454 25x25), variable: ALMTC.Level[iHMICbLevelSelection].AlarmID[15], style: Lamp-Lamp1-Red
    Label (444,454 40x25), "[ 15 ]:"
    Label (510,452 300x25), ": Debug Station Facility Ac Power OFF Detected"
    Lamp1 (486,481 25x25), variable: ALMTC.Level[iHMICbLevelSelection].AlarmID[16], style: Lamp-Lamp1-Red
    Label (444,481 40x25), "[ 16 ]:"
    Label (510,479 300x25), ": Front Side Door Lock Signal is not Detected"
    Lamp1 (486,508 25x25), variable: ALMTC.Level[iHMICbLevelSelection].AlarmID[17], style: Lamp-Lamp1-Red
    Label (444,508 40x25), "[ 17 ]:"
    Label (510,506 300x25), ": ipTCDrawerCylExtendRS signal not detected"
    Lamp1 (486,535 25x25), variable: ALMTC.Level[iHMICbLevelSelection].AlarmID[18], style: Lamp-Lamp1-Red
    Label (444,535 40x25), "[ 18 ]:"
    Label (510,533 300x25), ": ipTCDrawerCylRetractRS signal not detected"
    Lamp1 (486,562 25x25), variable: ALMTC.Level[iHMICbLevelSelection].AlarmID[19], style: Lamp-Lamp1-Red
    Label (444,562 40x25), "[ 19 ]:"
    Label (510,560 300x25), ": ipTCDrawerCylUp signal not detected"
    Lamp1 (486,589 25x25), variable: ALMTC.Level[iHMICbLevelSelection].AlarmID[20], style: Lamp-Lamp1-Red
    Label (444,589 40x25), "[ 20 ]:"
    Label (510,587 300x25), ": ipTCDrawerCylDown signal not detected"
    Lamp1 (66,80 25x25), variable: ALMTC.Common.AlarmID[1], style: Lamp-Lamp1-Red
    Label (24,80 40x25), "[ 01 ]:"
    Label (90,78 300x25), "Column PCW Leakage"
    Lamp1 (66,107 25x25), variable: ALMTC.Common.AlarmID[2], style: Lamp-Lamp1-Red
    Label (24,107 40x25), "[ 02 ]:"
    Label (90,105 300x25), "AllTCDrawer is not inside Cell"
    Lamp1 (66,134 25x25), variable: ALMTC.Common.AlarmID[3], style: Lamp-Lamp1-Red
    Label (24,134 40x25), "[ 03 ]:"
    Label (90,132 300x25), "ipTbotDoorClosedSignal not Detected"
    Lamp1 (66,161 25x25), variable: ALMTC.Common.AlarmID[4], style: Lamp-Lamp1-Red
    Label (24,161 40x25), "[ 04 ]:"
    Label (90,159 300x25), "---------"
    Label (587,25 81x40), "TESTER"
    Label (790,23 243x40), "ALARM ID BIT STATUS"
    Label (35,23 388x40), "TC COLUMN ALARM STATUS"
    Lamp1 (1242,78 25x25), style: Lamp-Lamp1-Yellow
    Label (1200,78 40x25), "[ P1]:"
    Label (1266,76 300x25), ": TIU UP SOLENOID"
    Lamp1 (1242,105 25x25), style: Lamp-Lamp1-Yellow
    Label (1200,105 40x25), "[ P2]:"
    Label (1266,103 300x25), ": TIU DOWN SOLENOID"
    Lamp1 (1242,132 25x25), style: Lamp-Lamp1-Yellow
    Label (1200,132 40x25), "[ P3]:"
    Label (1266,130 300x25), ": TIU EXTEND SOLENOID"
    Lamp1 (1242,159 25x25), style: Lamp-Lamp1-Yellow
    Label (1200,159 40x25), "[ P4]:"
    Label (1266,157 300x25), ": TIU RETRACT SOLENOID"
    Lamp1 (1242,186 25x25), style: Lamp-Lamp1-Yellow
    Label (1200,186 40x25), "[ P5]:"
    Label (1266,184 300x25), ": TIU EXTEND REED SWITCH"
    Lamp1 (1242,213 25x25), style: Lamp-Lamp1-Yellow
    Label (1200,213 40x25), "[ P6]:"
    Label (1266,211 300x25), ": TIU RETRACT REED SWITCH"
    Lamp1 (1242,240 25x25), variable: stEAP.stTBOT_TC_EAP[iHMICbLevelSelection].iTCDwrSafeToMoveEAP, style: Lamp-Lamp1-Yellow
    Label (1200,240 40x25), "[ S1]:"
    Label (1266,238 300x25), ": TIU NOT SAFETOMOVE (True:Not Safe,False: Safe)"
    Lamp1 (1242,267 25x25), variable: stEAP.stTBOT_TC_EAP[iHMICbLevelSelection].bAntiCollisionTriggered, style: Lamp-Lamp1-Yellow
    Label (1200,267 40x25), "[ S2]:"
    Label (1266,265 300x25), ": TBOT ANTI-COLLISION TRIGGERED SIGNAL"
    Lamp1 (1242,294 25x25), style: Lamp-Lamp1-Yellow
    Label (1200,294 40x25), "[ S3]:"
    Label (1266,292 300x25), ":(----------------------------------------------------------)"
    Lamp1 (1242,321 25x25), style: Lamp-Lamp1-Yellow
    Label (1200,321 40x25), "[ S4]:"
    Label (1266,319 300x25), ":(----------------------------------------------------------)"
    Lamp1 (1242,348 25x25), style: Lamp-Lamp1-Yellow
    Label (1200,348 40x25), "[ S5]:"
    Label (1266,346 300x25), ":(----------------------------------------------------------)"
    Lamp1 (1242,375 25x25), style: Lamp-Lamp1-Yellow
    Label (1200,375 40x25), "[ S6]:"
    Label (1266,373 300x25), ":(----------------------------------------------------------)"
    Label (1207,24 305x40), "EAP SAFTY SIGNAL STATUS"
    Rectangle (14,314 414x505)
    Rectangle (14,315 414x46)
    Label (35,318 388x40), "DEBUG COLUMN ALARM STATUS"
    Lamp1 (62,363 25x25), variable: ALM_DCCOL.AlarmID[1], style: Lamp-Lamp1-Red
    Label (20,363 40x25), "[ 01 ]:"
    Label (86,361 300x25), ": eSystemPCWLeakageAlarm"
    Lamp1 (62,390 25x25), variable: ALM_DCCOL.AlarmID[2], style: Lamp-Lamp1-Red
    Label (20,390 40x25), "[ 02 ]:"
    Label (86,388 300x25), ": eSystemPCWSupplyLeakageAlarm"
    Lamp1 (62,417 25x25), variable: ALM_DCCOL.AlarmID[3], style: Lamp-Lamp1-Red
    Label (20,417 40x25), "[ 03 ]:"
    Label (86,415 300x25), ": eSystemPCWReturnLeakageAlarm"
    Lamp1 (62,444 25x25), variable: ALM_DCCOL.AlarmID[4], style: Lamp-Lamp1-Red
    Label (20,444 40x25), "[ 04 ]:"
    Label (86,442 300x25), ": eCriticalCondensationAlarm"
    Lamp1 (62,471 25x25), variable: ALM_DCCOL.AlarmID[5], style: Lamp-Lamp1-Red
    Label (20,471 40x25), "[ 05 ]:"
    Label (86,469 300x25), ": e6BarLowOFAAirPressureAlarm"
    Lamp1 (62,498 25x25), variable: ALM_DCCOL.AlarmID[6], style: Lamp-Lamp1-Red
    Label (20,498 40x25), "[ 06 ]:"
    Label (86,496 300x25), ": eSystemPCWLeakage2Alarm"
    Lamp1 (62,525 25x25), variable: ALM_DCCOL.AlarmID[7], style: Lamp-Lamp1-Red
    Label (20,525 40x25), "[ 07 ]:"
    Label (86,523 300x25), ":(--------------------------------------------------------------)"
    Lamp1 (62,552 25x25), variable: ALM_DCCOL.AlarmID[8], style: Lamp-Lamp1-Red
    Label (20,552 40x25), "[ 08 ]:"
    Label (86,550 300x25), ":(--------------------------------------------------------------)"
    Lamp1 (62,579 25x25), variable: ALM_DCCOL.AlarmID[9], style: Lamp-Lamp1-Red
    Label (20,579 40x25), "[ 09 ]:"
    Label (86,577 300x25), ":(--------------------------------------------------------------)"
    Lamp1 (62,606 25x25), variable: ALM_DCCOL.AlarmID[10], style: Lamp-Lamp1-Red
    Label (20,606 40x25), "[ 10 ]:"
    Label (86,604 300x25), ":(--------------------------------------------------------------)"
    Lamp1 (62,633 25x25), variable: ALM_DCCOL.AlarmID[11], style: Lamp-Lamp1-Red
    Label (20,633 40x25), "[ 11 ]:"
    Label (86,631 300x25), ": ePCWSupplyHighTempWarning"
    Lamp1 (62,660 25x25), variable: ALM_DCCOL.AlarmID[12], style: Lamp-Lamp1-Red
    Label (20,660 40x25), "[ 12 ]:"
    Label (86,658 300x25), ": e6BarLowOFAAirPressureWarning"
    Lamp1 (62,687 25x25), variable: ALM_DCCOL.AlarmID[13], style: Lamp-Lamp1-Red
    Label (20,687 40x25), "[ 13 ]:"
    Label (86,685 300x25), ": e9BarLowOFAAirPressureWarning"
    Lamp1 (62,714 25x25), variable: ALM_DCCOL.AlarmID[14], style: Lamp-Lamp1-Red
    Label (20,714 40x25), "[ 14 ]:"
    Label (86,712 300x25), ": eExcessiveHeatLoadIntoPCWWarning"
    Lamp1 (62,741 25x25), variable: ALM_DCCOL.AlarmID[15], style: Lamp-Lamp1-Red
    Label (20,741 40x25), "[ 15 ]:"
    Label (86,739 300x25), ": eCondensationWarning"
    Lamp1 (62,768 25x25), variable: ALM_DCCOL.AlarmID[16], style: Lamp-Lamp1-Red
    Label (20,768 40x25), "[ 16 ]:"
    Label (86,766 300x25), ":(--------------------------------------------------------------)"
    Lamp1 (62,795 25x25), variable: ALM_DCCOL.AlarmID[17], style: Lamp-Lamp1-Red
    Label (20,795 40x25), "[ 17 ]:"
    Label (86,793 300x25), ":(--------------------------------------------------------------)"
    RoundedRectangle (89,832 200x25), "DBColumnPCWLeakageEAP"
        toggle fbDebugColumn.stDebugColumnDIO.eapDBColumnPCWLeakage
    Lamp1 (60,830 30x30), variable: fbDebugColumn.stDebugColumnDIO.eapDBColumnPCWLeakage, style: Lamp-Lamp1-Green
    RoundedRectangle (89,862 200x25), "DBColumnPCWSupplyLeakageEAP"
        toggle fbDebugColumn.stDebugColumnDIO.eapDBColumnPCWSupplyLeakage
    Lamp1 (60,860 30x30), variable: fbDebugColumn.stDebugColumnDIO.eapDBColumnPCWSupplyLeakage, style: Lamp-Lamp1-Green
    RoundedRectangle (89,892 200x25), "DBColumnPCWReturnLeakageEAP"
        toggle fbDebugColumn.stDebugColumnDIO.eapDBColumnPCWReturnLeakage
    Lamp1 (60,890 30x30), variable: fbDebugColumn.stDebugColumnDIO.eapDBColumnPCWReturnLeakage, style: Lamp-Lamp1-Green
    Frame (1577,19 355x2000), invisible if: Not bEnableManualCommandTest1 AND Not bEnableManualCommandTest2
        shows HMI_ManualCommand()
END_VISUALIZATION

// ---- VISUs/HMI_DebugCell_Stack.TcVIS
VISUALIZATION HMI_DebugCell_Stack  // 2x2
END_VISUALIZATION

// ---- VISUs/HMI_DebugStation.TcVIS
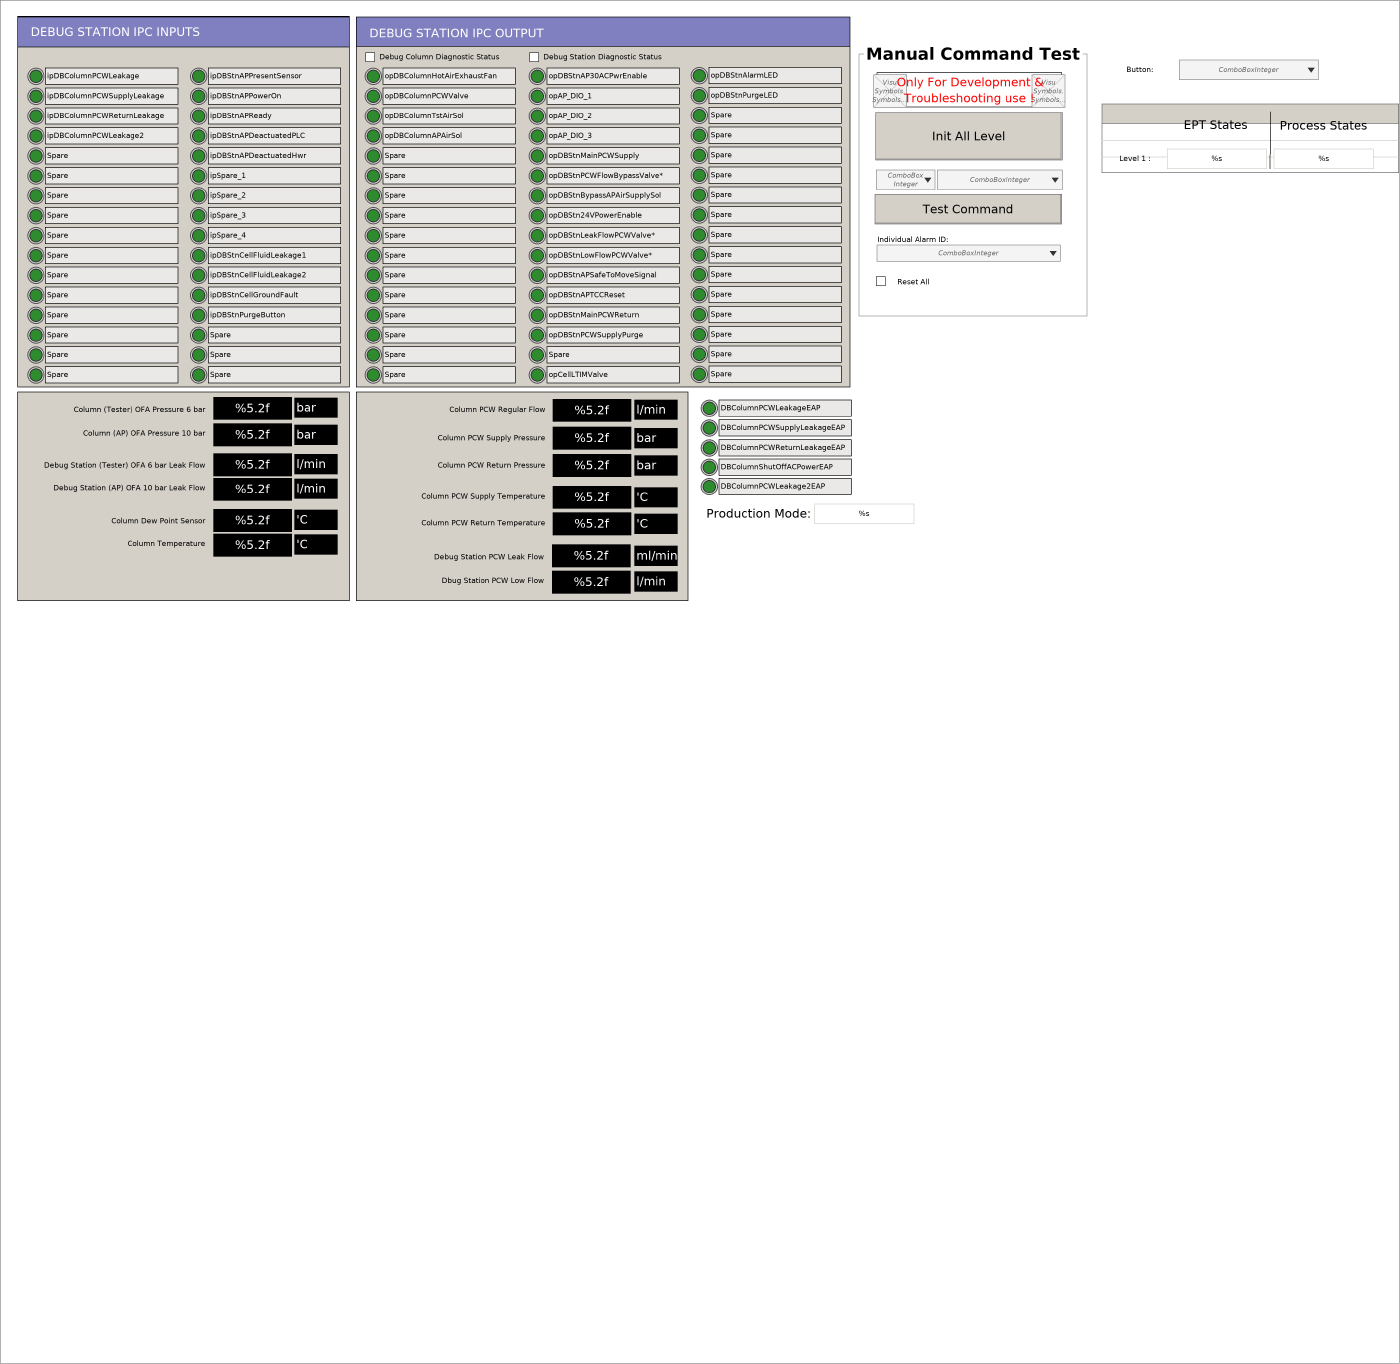
VISUALIZATION HMI_DebugStation  // 2108x2055
    Rectangle (536,590 500x315)
    Rectangle (26,590 500x315)
    Rectangle (536,42 744x541)
    Rectangle (536,25 744x45)
    Label (553,30 500x40), "DEBUG STATION IPC OUTPUT"
    Rectangle (26,24 500x559)
    Rectangle (26,25 500x46)
    Label (43,28 500x40), "DEBUG STATION IPC INPUTS"
    RoundedRectangle (68,102 200x25), "ipDBColumnPCWLeakage"
    Lamp1 (39,100 30x30), variable: fbDebugColumn.stDebugColumnDIO.ipDBColumnPCWLeakage, style: Lamp-Lamp1-Green
    RoundedRectangle (576,102 200x25), "opDBColumnHotAirExhaustFan"
        toggle fbDebugColumn.stDebugColumnDIO.opDBColumnHotAirExhaustFan
    Lamp1 (547,100 30x30), variable: fbDebugColumn.stDebugColumnDIO.opDBColumnHotAirExhaustFan, style: Lamp-Lamp1-Green
    RoundedRectangle (68,132 200x25), "ipDBColumnPCWSupplyLeakage"
    Lamp1 (39,130 30x30), variable: fbDebugColumn.stDebugColumnDIO.ipDBColumnPCWSupplyLeakage, style: Lamp-Lamp1-Green
    RoundedRectangle (68,162 200x25), "ipDBColumnPCWReturnLeakage"
    Lamp1 (39,160 30x30), variable: fbDebugColumn.stDebugColumnDIO.ipDBColumnPCWReturnLeakage, style: Lamp-Lamp1-Green
    RoundedRectangle (68,192 200x25), "ipDBColumnPCWLeakage2"
    Lamp1 (39,190 30x30), variable: fbDebugColumn.stDebugColumnDIO.ipDBColumnPCWLeakage2, style: Lamp-Lamp1-Green
    RoundedRectangle (68,222 200x25), "Spare"
    Lamp1 (39,220 30x30), style: Lamp-Lamp1-Green
    RoundedRectangle (68,252 200x25), "Spare"
    Lamp1 (39,250 30x30), style: Lamp-Lamp1-Green
    RoundedRectangle (68,282 200x25), "Spare"
    Lamp1 (39,280 30x30), style: Lamp-Lamp1-Green
    RoundedRectangle (68,312 200x25), "Spare"
    Lamp1 (39,310 30x30), style: Lamp-Lamp1-Green
    RoundedRectangle (68,342 200x25), "Spare"
    Lamp1 (39,340 30x30), style: Lamp-Lamp1-Green
    RoundedRectangle (68,372 200x25), "Spare"
    Lamp1 (39,370 30x30), style: Lamp-Lamp1-Green
    RoundedRectangle (68,402 200x25), "Spare"
    Lamp1 (39,400 30x30), style: Lamp-Lamp1-Green
    RoundedRectangle (68,432 200x25), "Spare"
    Lamp1 (39,430 30x30), style: Lamp-Lamp1-Green
    RoundedRectangle (68,462 200x25), "Spare"
    Lamp1 (39,460 30x30), style: Lamp-Lamp1-Green
    RoundedRectangle (68,492 200x25), "Spare"
    Lamp1 (39,490 30x30), style: Lamp-Lamp1-Green
    RoundedRectangle (68,522 200x25), "Spare"
    Lamp1 (39,520 30x30), style: Lamp-Lamp1-Green
    RoundedRectangle (68,552 200x25), "Spare"
    Lamp1 (39,550 30x30), style: Lamp-Lamp1-Green
    RoundedRectangle (576,132 200x25), "opDBColumnPCWValve"
        toggle fbDebugColumn.stDebugColumnDIO.opDBColumnPCWValve
    Lamp1 (547,130 30x30), variable: fbDebugColumn.stDebugColumnDIO.opDBColumnPCWValve, style: Lamp-Lamp1-Green
    RoundedRectangle (576,162 200x25), "opDBColumnTstAirSol"
        toggle fbDebugColumn.stDebugColumnDIO.opDBColumnTstAirSol
    Lamp1 (547,160 30x30), variable: fbDebugColumn.stDebugColumnDIO.opDBColumnTstAirSol, style: Lamp-Lamp1-Green
    RoundedRectangle (576,192 200x25), "opDBColumnAPAirSol"
        toggle fbDebugColumn.stDebugColumnDIO.opDBColumnAPAirSol
    Lamp1 (547,190 30x30), variable: fbDebugColumn.stDebugColumnDIO.opDBColumnAPAirSol, style: Lamp-Lamp1-Green
    RoundedRectangle (576,222 200x25), "Spare"
    Lamp1 (547,220 30x30), style: Lamp-Lamp1-Green
    RoundedRectangle (576,252 200x25), "Spare"
    Lamp1 (547,250 30x30), style: Lamp-Lamp1-Green
    RoundedRectangle (576,282 200x25), "Spare"
    Lamp1 (547,280 30x30), style: Lamp-Lamp1-Green
    RoundedRectangle (576,312 200x25), "Spare"
    Lamp1 (547,310 30x30), style: Lamp-Lamp1-Green
    RoundedRectangle (576,342 200x25), "Spare"
    Lamp1 (547,340 30x30), style: Lamp-Lamp1-Green
    RoundedRectangle (576,372 200x25), "Spare"
    Lamp1 (547,370 30x30), style: Lamp-Lamp1-Green
    RoundedRectangle (576,402 200x25), "Spare"
    Lamp1 (547,400 30x30), style: Lamp-Lamp1-Green
    RoundedRectangle (576,432 200x25), "Spare"
    Lamp1 (547,430 30x30), style: Lamp-Lamp1-Green
    RoundedRectangle (576,462 200x25), "Spare"
    Lamp1 (547,460 30x30), style: Lamp-Lamp1-Green
    RoundedRectangle (576,492 200x25), "Spare"
    Lamp1 (547,490 30x30), style: Lamp-Lamp1-Green
    RoundedRectangle (576,522 200x25), "Spare"
    Lamp1 (547,520 30x30), style: Lamp-Lamp1-Green
    RoundedRectangle (576,552 200x25), "Spare"
    Lamp1 (547,550 30x30), style: Lamp-Lamp1-Green
    RoundedRectangle (313,102 200x25), "ipDBStnAPPresentSensor"
    Lamp1 (284,100 30x30), variable: stDebugStation.fbDBStnSeq.stDebugStationDIO.ipDBStnAPPresentSensor, style: Lamp-Lamp1-Green
    RoundedRectangle (313,132 200x25), "ipDBStnAPPowerOn"
    Lamp1 (284,130 30x30), variable: stDebugStation.fbDBStnSeq.stDebugStationDIO.ipDBStnAPPowerOn, style: Lamp-Lamp1-Green
    RoundedRectangle (313,162 200x25), "ipDBStnAPReady"
    Lamp1 (284,160 30x30), variable: stDebugStation.fbDBStnSeq.stDebugStationDIO.ipDBStnAPReady, style: Lamp-Lamp1-Green
    RoundedRectangle (313,192 200x25), "ipDBStnAPDeactuatedPLC"
    Lamp1 (284,190 30x30), variable: stDebugStation.fbDBStnSeq.stDebugStationDIO.ipDBStnHandlerSafeToEnterPLC, style: Lamp-Lamp1-Green
    RoundedRectangle (313,222 200x25), "ipDBStnAPDeactuatedHwr"
    Lamp1 (284,220 30x30), variable: stDebugStation.fbDBStnSeq.stDebugStationDIO.ipDBStnHandlerSafeToEnterHwr, style: Lamp-Lamp1-Green
    RoundedRectangle (313,252 200x25), "ipSpare_1"
    Lamp1 (284,250 30x30), variable: stDebugStation.fbDBStnSeq.stDebugStationDIO.ipSpare_1, style: Lamp-Lamp1-Green
    RoundedRectangle (313,282 200x25), "ipSpare_2"
    Lamp1 (284,280 30x30), variable: stDebugStation.fbDBStnSeq.stDebugStationDIO.ipSpare_2, style: Lamp-Lamp1-Green
    RoundedRectangle (313,312 200x25), "ipSpare_3"
    Lamp1 (284,310 30x30), variable: stDebugStation.fbDBStnSeq.stDebugStationDIO.ipSpare_3, style: Lamp-Lamp1-Green
    RoundedRectangle (313,342 200x25), "ipSpare_4"
    Lamp1 (284,340 30x30), variable: stDebugStation.fbDBStnSeq.stDebugStationDIO.ipSpare_4, style: Lamp-Lamp1-Green
    RoundedRectangle (313,372 200x25), "ipDBStnCellFluidLeakage1"
    Lamp1 (284,370 30x30), variable: stDebugStation.fbDBStnSeq.stDebugStationDIO.ipDBStnCellFluidLeakage1, style: Lamp-Lamp1-Green
    RoundedRectangle (313,402 200x25), "ipDBStnCellFluidLeakage2"
    Lamp1 (284,400 30x30), variable: stDebugStation.fbDBStnSeq.stDebugStationDIO.ipDBStnCellFluidLeakage2, style: Lamp-Lamp1-Green
    RoundedRectangle (313,432 200x25), "ipDBStnCellGroundFault"
    Lamp1 (284,430 30x30), variable: stDebugStation.fbDBStnSeq.stDebugStationDIO.ipDBStnCellGroundFault, style: Lamp-Lamp1-Green
    RoundedRectangle (313,462 200x25), "ipDBStnPurgeButton"
    Lamp1 (284,460 30x30), variable: stDebugStation.fbDBStnSeq.stDebugStationDIO.ipDBStnPurgeButton, style: Lamp-Lamp1-Green
    RoundedRectangle (313,492 200x25), "Spare"
    Lamp1 (284,490 30x30), style: Lamp-Lamp1-Green
    RoundedRectangle (313,522 200x25), "Spare"
    Lamp1 (284,520 30x30), style: Lamp-Lamp1-Green
    RoundedRectangle (313,552 200x25), "Spare"
    Lamp1 (284,550 30x30), style: Lamp-Lamp1-Green
    RoundedRectangle (823,102 200x25), "opDBStnAP30ACPwrEnable"
        toggle stDebugStation.fbDBStnSeq.stDebugStationDIO.opDBStnAP240ACPwrEnable
    Lamp1 (794,100 30x30), variable: stDebugStation.fbDBStnSeq.stDebugStationDIO.opDBStnAP240ACPwrEnable, style: Lamp-Lamp1-Green
    RoundedRectangle (823,132 200x25), "opAP_DIO_1"
        toggle stDebugStation.fbDBStnSeq.stDebugStationDIO.opAP_DIO_1
    Lamp1 (794,130 30x30), variable: stDebugStation.fbDBStnSeq.stDebugStationDIO.opAP_DIO_1, style: Lamp-Lamp1-Green
    RoundedRectangle (823,162 200x25), "opAP_DIO_2"
        toggle stDebugStation.fbDBStnSeq.stDebugStationDIO.opAP_DIO_2
    Lamp1 (794,160 30x30), variable: stDebugStation.fbDBStnSeq.stDebugStationDIO.opAP_DIO_2, style: Lamp-Lamp1-Green
    RoundedRectangle (823,192 200x25), "opAP_DIO_3"
        toggle stDebugStation.fbDBStnSeq.stDebugStationDIO.opAP_DIO_3
    Lamp1 (794,190 30x30), variable: stDebugStation.fbDBStnSeq.stDebugStationDIO.opAP_DIO_3, style: Lamp-Lamp1-Green
    RoundedRectangle (823,222 200x25), "opDBStnMainPCWSupply"
        toggle stDebugStation.fbDBStnSeq.stDebugStationDIO.opDBStnPCWValve
    Lamp1 (794,220 30x30), variable: stDebugStation.fbDBStnSeq.stDebugStationDIO.opDBStnPCWValve, style: Lamp-Lamp1-Green
    RoundedRectangle (823,252 200x25), "opDBStnPCWFlowBypassValve*"
        toggle stDebugStation.fbDBStnSeq.stDebugStationDIO.opDBStnPCWFlowBypassValve
    Lamp1 (794,250 30x30), variable: stDebugStation.fbDBStnSeq.stDebugStationDIO.opDBStnPCWFlowBypassValve, style: Lamp-Lamp1-Green
    RoundedRectangle (823,282 200x25), "opDBStnBypassAPAirSupplySol"
        toggle stDebugStation.fbDBStnSeq.stDebugStationDIO.opDBStnBypassAPAirSupplySol
    Lamp1 (794,280 30x30), variable: stDebugStation.fbDBStnSeq.stDebugStationDIO.opDBStnBypassAPAirSupplySol, style: Lamp-Lamp1-Green
    RoundedRectangle (823,312 200x25), "opDBStn24VPowerEnable"
        toggle stDebugStation.fbDBStnSeq.stDebugStationDIO.opDBStn24VPowerEnable
    Lamp1 (794,310 30x30), variable: stDebugStation.fbDBStnSeq.stDebugStationDIO.opDBStn24VPowerEnable, style: Lamp-Lamp1-Green
    RoundedRectangle (823,342 200x25), "opDBStnLeakFlowPCWValve*"
        toggle stDebugStation.fbDBStnSeq.stDebugStationDIO.opDBStnLeakFlowPCWValve
    Lamp1 (794,340 30x30), variable: stDebugStation.fbDBStnSeq.stDebugStationDIO.opDBStnLeakFlowPCWValve, style: Lamp-Lamp1-Green
    RoundedRectangle (823,372 200x25), "opDBStnLowFlowPCWValve*"
        toggle stDebugStation.fbDBStnSeq.stDebugStationDIO.opDBStnLowFlowPCWValve
    Lamp1 (794,370 30x30), variable: stDebugStation.fbDBStnSeq.stDebugStationDIO.opDBStnLowFlowPCWValve, style: Lamp-Lamp1-Green
    RoundedRectangle (823,402 200x25), "opDBStnAPSafeToMoveSignal"
        toggle stDebugStation.fbDBStnSeq.stDebugStationDIO.opDBStnAPSafeToEngage
    Lamp1 (794,400 30x30), variable: stDebugStation.fbDBStnSeq.stDebugStationDIO.opDBStnAPSafeToEngage, style: Lamp-Lamp1-Green
    RoundedRectangle (823,432 200x25), "opDBStnAPTCCReset"
        toggle stDebugStation.fbDBStnSeq.stDebugStationDIO.opDBStnAPTCCReset
    Lamp1 (794,430 30x30), variable: stDebugStation.fbDBStnSeq.stDebugStationDIO.opDBStnAPTCCReset, style: Lamp-Lamp1-Green
    RoundedRectangle (823,462 200x25), "opDBStnMainPCWReturn"
        toggle stDebugStation.fbDBStnSeq.stDebugStationDIO.opDBStnMainPCWReturn
    Lamp1 (794,460 30x30), variable: stDebugStation.fbDBStnSeq.stDebugStationDIO.opDBStnMainPCWReturn, style: Lamp-Lamp1-Green
    RoundedRectangle (823,492 200x25), "opDBStnPCWSupplyPurge"
        toggle stDebugStation.fbDBStnSeq.stDebugStationDIO.opDBStnPCWSupplyPurge
    Lamp1 (794,490 30x30), variable: stDebugStation.fbDBStnSeq.stDebugStationDIO.opDBStnPCWSupplyPurge, style: Lamp-Lamp1-Green
    RoundedRectangle (823,522 200x25), "Spare"
    Lamp1 (794,520 30x30), style: Lamp-Lamp1-Green
    RoundedRectangle (823,552 200x25), "opCellLTIMValve"
        toggle stDebugStation.fbDBStnSeq.stDebugStationDIO.opCellLTIMValve
    Lamp1 (794,550 30x30), variable: stDebugStation.fbDBStnSeq.stDebugStationDIO.opCellLTIMValve, style: Lamp-Lamp1-Green
    Textfield (320,597 120x36), "%5.2f", text variable: fbDebugColumn.stDebugColumnDIO.ipDBColumnTstAirPressure, input disabled if: TRUE
    Textfield (320,637 120x36), "%5.2f", text variable: fbDebugColumn.stDebugColumnDIO.ipDBColumnAPAirPressure, input disabled if: TRUE
    Textfield (320,682 120x36), "%5.2f", text variable: stDebugStation.fbDBStnSeq.stDebugStationDIO.ipDBStnTstAirLeakFlowSensor, input disabled if: TRUE
    Textfield (320,719 120x36), "%5.2f", text variable: stDebugStation.fbDBStnSeq.stDebugStationDIO.ipDBStnAPAirLeakFlowSensor, input disabled if: TRUE
    Label (51,686 261x30), "Debug Station (Tester) OFA 6 bar Leak Flow"
    Label (44,720 268x30), "Debug Station (AP) OFA 10 bar Leak Flow"
    Label (60,602 252x30), "Column (Tester) OFA Pressure 6 bar"
    Label (81,638 231x30), "Column (AP) OFA Pressure 10 bar"
    Textfield (830,819 120x36), "%5.2f", text variable: stDebugStation.fbDBStnSeq.stDebugStationDIO.ipDBStnPCWLeakFlowSensor, input disabled if: TRUE
    Textfield (830,859 120x36), "%5.2f", text variable: stDebugStation.fbDBStnSeq.stDebugStationDIO.ipDBStnPCWLowFlowSensor, input disabled if: TRUE
    Label (620,824 202x30), "Debug Station PCW Leak Flow"
    Label (574,860 248x30), "Dbug Station PCW Low Flow"
    Textfield (831,771 120x36), "%5.2f", text variable: fbDebugColumn.stDebugColumnDIO.ipDBColumnPCWReturnTemperature, input disabled if: TRUE
    Textfield (831,683 120x36), "%5.2f", text variable: fbDebugColumn.stDebugColumnDIO.ipDBColumnPCWReturnPressure, input disabled if: TRUE
    Textfield (831,600 120x36), "%5.2f", text variable: fbDebugColumn.stDebugColumnDIO.ipDBColumnPCWRegularFlowSensor, input disabled if: TRUE
    Textfield (831,642 120x36), "%5.2f", text variable: fbDebugColumn.stDebugColumnDIO.ipDBColumnPCWSupplyPressure, input disabled if: TRUE
    Textfield (831,731 120x36), "%5.2f", text variable: fbDebugColumn.stDebugColumnDIO.ipDBColumnPCWSupplyTemperature, input disabled if: TRUE
    Label (613,602 211x30), "Column PCW Regular Flow"
    Label (616,645 208x30), "Column PCW Supply Pressure"
    Label (641,686 183x30), "Column PCW Return Pressure"
    Label (595,733 229x30), "Column PCW Supply Temperature"
    Label (611,773 213x30), "Column PCW Return Temperature"
    Rectangle (955,602 65x30), "l/min"
    Rectangle (955,645 65x30), "bar"
    Rectangle (955,686 65x30), "bar"
    Rectangle (955,734 65x30), "'C"
    Rectangle (955,774 65x30), "'C"
    Rectangle (955,822 65x30), "ml/min"
    Rectangle (955,861 65x30), "l/min"
    Rectangle (443,599 65x30), "bar"
    Rectangle (443,640 65x30), "bar"
    Rectangle (443,684 65x30), "l/min"
    Rectangle (443,721 65x30), "l/min"
    Textfield (320,766 120x36), "%5.2f", text variable: fbDebugColumn.stDebugColumnDIO.ipDBColumnDewPointSensor, input disabled if: TRUE
    Textfield (320,803 120x36), "%5.2f", text variable: fbDebugColumn.stDebugColumnDIO.ipDBColumnTempSensor, input disabled if: TRUE
    Label (133,770 179x30), "Column Dew Point Sensor"
    Label (162,804 150x30), "Column Temperature"
    Rectangle (443,768 65x30), "'C"
    Rectangle (443,805 65x30), "'C"
    Checkbox (795,71 224x30), "Debug Station Diagnostic Status", variable: stDebugStation.fbDBStnSeq.stDebugStationVIO.bDiagnosticMode
    Checkbox (548,71 222x30), "Debug Column Diagnostic Status", variable: fbDebugColumn.stDebugColumnVIO.bDiagnosticMode
    RoundedRectangle (1082,602 200x25), "DBColumnPCWLeakageEAP"
        toggle fbDebugColumn.stDebugColumnDIO.eapDBColumnPCWLeakage
    Lamp1 (1053,600 30x30), variable: fbDebugColumn.stDebugColumnDIO.eapDBColumnPCWLeakage, style: Lamp-Lamp1-Green
    RoundedRectangle (1082,632 200x25), "DBColumnPCWSupplyLeakageEAP"
        toggle fbDebugColumn.stDebugColumnDIO.eapDBColumnPCWSupplyLeakage
    Lamp1 (1053,630 30x30), variable: fbDebugColumn.stDebugColumnDIO.eapDBColumnPCWSupplyLeakage, style: Lamp-Lamp1-Green
    RoundedRectangle (1082,662 200x25), "DBColumnPCWReturnLeakageEAP"
        toggle fbDebugColumn.stDebugColumnDIO.eapDBColumnPCWReturnLeakage
    Lamp1 (1053,660 30x30), variable: fbDebugColumn.stDebugColumnDIO.eapDBColumnPCWReturnLeakage, style: Lamp-Lamp1-Green
    Frame (1284,53 355x2000), invisible if: Not bEnableManualCommandTest1 AND Not bEnableManualCommandTest2
        shows HMI_ManualCommand()
    Lamp1 (1038,99 30x30), variable: stDebugStation.fbDBStnSeq.stDebugStationDIO.opDBStnAlarmLED, style: Lamp-Lamp1-Green
    RoundedRectangle (1067,101 200x25), "opDBStnAlarmLED"
        toggle stDebugStation.fbDBStnSeq.stDebugStationDIO.opDBStnAlarmLED
    RoundedRectangle (1067,131 200x25), "opDBStnPurgeLED"
        toggle stDebugStation.fbDBStnSeq.stDebugStationDIO.opDBStnPurgeLED
    Lamp1 (1038,129 30x30), variable: stDebugStation.fbDBStnSeq.stDebugStationDIO.opDBStnPurgeLED, style: Lamp-Lamp1-Green
    RoundedRectangle (1067,161 200x25), "Spare"
    Lamp1 (1038,159 30x30), style: Lamp-Lamp1-Green
    RoundedRectangle (1067,191 200x25), "Spare"
    Lamp1 (1038,189 30x30), style: Lamp-Lamp1-Green
    RoundedRectangle (1067,221 200x25), "Spare"
    Lamp1 (1038,219 30x30), style: Lamp-Lamp1-Green
    RoundedRectangle (1067,251 200x25), "Spare"
    Lamp1 (1038,249 30x30), style: Lamp-Lamp1-Green
    RoundedRectangle (1067,281 200x25), "Spare"
    Lamp1 (1038,279 30x30), style: Lamp-Lamp1-Green
    RoundedRectangle (1067,311 200x25), "Spare"
    Lamp1 (1038,309 30x30), style: Lamp-Lamp1-Green
    RoundedRectangle (1067,341 200x25), "Spare"
    Lamp1 (1038,339 30x30), style: Lamp-Lamp1-Green
    RoundedRectangle (1067,371 200x25), "Spare"
    Lamp1 (1038,369 30x30), style: Lamp-Lamp1-Green
    RoundedRectangle (1067,401 200x25), "Spare"
    Lamp1 (1038,399 30x30), style: Lamp-Lamp1-Green
    RoundedRectangle (1067,431 200x25), "Spare"
    Lamp1 (1038,429 30x30), style: Lamp-Lamp1-Green
    RoundedRectangle (1067,461 200x25), "Spare"
    Lamp1 (1038,459 30x30), style: Lamp-Lamp1-Green
    RoundedRectangle (1067,491 200x25), "Spare"
    Lamp1 (1038,489 30x30), style: Lamp-Lamp1-Green
    RoundedRectangle (1067,521 200x25), "Spare"
    Lamp1 (1038,519 30x30), style: Lamp-Lamp1-Green
    RoundedRectangle (1067,551 200x25), "Spare"
    Lamp1 (1038,549 30x30), style: Lamp-Lamp1-Green
    RoundedRectangle (1082,691 200x25), "DBColumnShutOffACPowerEAP"
        toggle fbDebugColumn.stDebugColumnDIO.eapShutOffAllACPower
    Lamp1 (1053,689 30x30), variable: fbDebugColumn.stDebugColumnDIO.eapShutOffAllACPower, style: Lamp-Lamp1-Green
    ComboBoxInteger (1775,90 210x30), variable: TestManually.iBtnNo, text list: 'BtnTxtList'
    Label (1680,90 76x30), "Button:"
    RoundedRectangle (1082,720 200x25), "DBColumnPCWLeakage2EAP"
        toggle fbDebugColumn.stDebugColumnDIO.eapDBColumnPCWLeakage2
    Lamp1 (1053,718 30x30), variable: fbDebugColumn.stDebugColumnDIO.eapDBColumnPCWLeakage2, style: Lamp-Lamp1-Green
    Label (1065,759 160x30), "Production Mode:"
    Textfield (1226,759 150x30), "%s", text variable: bProductionMode
    Table (1659,156 447x104)
    Label (1671,224 80x30), "Level 1 :"
    Textfield (1757,224 150x30), "%s", text variable: TC_EPT[1].TCSite[1].TCU
    Label (1755,170 151x37), "EPT States"
    Textfield (1918,224 150x30), "%s", text variable: stDebugStation.stGblDBStnParam.iProcessState
    Label (1914,171 158x37), "Process States"
    Line (1913,168) (1912,254)
END_VISUALIZATION

// ---- VISUs/HMI_FacilityAlarm_OFADewpoint.TcVIS
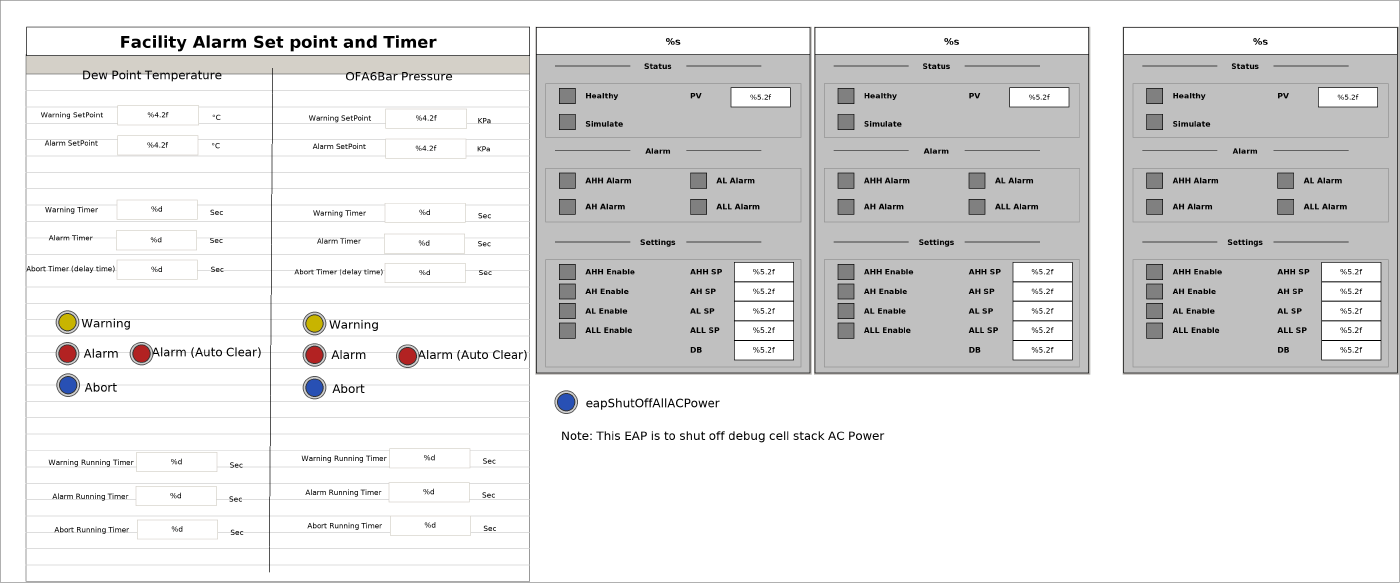
VISUALIZATION HMI_FacilityAlarm_OFADewpoint  // 2136x891
    Table (39,83 769x806)
    Rectangle (40,41 768x44)
    Label (48,49 753x30), "Facility Alarm Set point and Timer"
    Label (41,90 382x50), "Dew Point Temperature"
    Label (421,92 376x50), "OFA6Bar Pressure"
    Textfield (179,161 124x30), "%4.2f", text variable: DewPoint_LowSP
        OnMouseClick: write DewPoint_LowSP via Default
    Label (44,161 132x30), "Warning SetPoint"
    Label (308,165 44x30), "°C"
    Label (43,204 132x30), "Alarm SetPoint"
    Textfield (179,207 123x30), "%4.2f", text variable: DewPoint_LowLowSP
        OnMouseClick: write DewPoint_LowLowSP via Default
    Label (307,208 44x30), "°C"
    Textfield (178,305 123x30), "%d", text variable: DewPoint_Warning_Timer
        OnMouseClick: write DewPoint_Warning_Timer via Default
    Label (42,306 134x30), "Warning Timer"
    Label (306,310 49x30), "Sec"
    Textfield (177,352 123x30), "%d", text variable: DewPoint_Alarm_Timer
        OnMouseClick: write DewPoint_Alarm_Timer via Default
    Label (41,349 134x30), "Alarm Timer"
    Label (305,353 50x30), "Sec"
    Textfield (178,397 123x30), "%d", text variable: DewPoint_Abort_Timer
        OnMouseClick: write DewPoint_Abort_Timer via Default
    Label (42,396 132x30), "Abort Timer (delay time)"
    Label (305,397 53x30), "Sec"
    Label (453,166 132x30), "Warning SetPoint"
    Textfield (588,166 124x30), "%4.2f", text variable: OFA6Bar_LowSP
        OnMouseClick: write OFA6Bar_LowSP via Default
    Label (717,170 44x30), "KPa"
    Label (452,209 132x30), "Alarm SetPoint"
    Textfield (588,212 123x30), "%4.2f", text variable: OFA6Bar_LowLowSP
        OnMouseClick: write OFA6Bar_LowLowSP via Default
    Label (716,213 44x30), "KPa"
    Textfield (587,310 123x30), "%d", text variable: OFA6Bar_Warning_Timer
        OnMouseClick: write OFA6Bar_Warning_Timer via Default
    Label (451,311 134x30), "Warning Timer"
    Label (715,315 49x30), "Sec"
    Textfield (586,357 123x30), "%d", text variable: OFA6Bar_Alarm_Timer
        OnMouseClick: write OFA6Bar_Alarm_Timer via Default
    Label (450,354 134x30), "Alarm Timer"
    Label (714,358 50x30), "Sec"
    Textfield (587,402 123x30), "%d", text variable: OFA6Bar_Abort_Timer
        OnMouseClick: write OFA6Bar_Abort_Timer via Default
    Label (451,401 132x30), "Abort Timer (delay time)"
    Label (714,402 53x30), "Sec"
    Frame (817,41 421x531)
        shows AIN_Template(DUT := fbDebugColumn.fb_facility_DewPoint_OFA6Bar._DUT_AIN_InletTemp)
    Frame (1242,41 421x531)
        shows AIN_Template(DUT := fbDebugColumn.fb_facility_DewPoint_OFA6Bar._DUT_AIN_DewPoint)
    Frame (1713,41 421x531)
        shows AIN_Template(DUT := fbDebugColumn.fb_facility_DewPoint_OFA6Bar._DUT_AIN_6BarOFA)
    Lamp1 (77,472 52x41), variable: ALM_DCCOL.AlarmID[15], style: Lamp-Lamp1-Yellow
    Lamp1 (77,520 52x41), variable: ALM_DCCOL.AlarmID[4], style: Lamp-Lamp1-Red
    Lamp1 (454,522 52x41), variable: ALM_DCCOL.AlarmID[5], style: Lamp-Lamp1-Red
    Lamp1 (454,474 52x41), variable: ALM_DCCOL.AlarmID[12], style: Lamp-Lamp1-Yellow
    Label (491,480 98x33), "Warning"
    Label (493,526 79x33), "Alarm"
    Lamp1 (454,572 52x41), variable: OFA6Bar_Abort, style: Lamp-Lamp1-Blue
    Label (491,578 82x33), "Abort"
    Lamp1 (78,568 52x41), variable: DewPoint_Abort, style: Lamp-Lamp1-Blue
    Lamp1 (838,594 52x41), variable: fbDebugColumn.stDebugColumnDIO.eapShutOffAllACPower, style: Lamp-Lamp1-Blue
    Label (875,600 242x33), "eapShutOffAllACPower"
    Label (824,650 557x33), "Note: This EAP is to shut off debug cell stack AC Power"
    Label (113,478 98x33), "Warning"
    Label (115,524 79x33), "Alarm"
    Label (113,576 82x33), "Abort"
    Label (635,526 173x33), "Alarm (Auto Clear)"
    Lamp1 (596,524 52x41), variable: OFA6Bar_Alarm, style: Lamp-Lamp1-Red
    Label (229,522 173x33), "Alarm (Auto Clear)"
    Lamp1 (190,520 52x41), variable: DewPoint_Alarm, style: Lamp-Lamp1-Red
    Textfield (594,685 123x30), "%d", text variable: fbDebugColumn.fb_facility_DewPoint_OFA6Bar.fb_6BarOFA_Alarm._WarningStateTimer
    Label (458,686 134x30), "Warning Running Timer"
    Label (722,690 49x30), "Sec"
    Textfield (593,737 123x30), "%d", text variable: fbDebugColumn.fb_facility_DewPoint_OFA6Bar.fb_6BarOFA_Alarm._AlarmStateTimer
    Label (457,738 134x30), "Alarm Running Timer"
    Label (721,742 49x30), "Sec"
    Textfield (595,788 123x30), "%d", text variable: fbDebugColumn.fb_facility_DewPoint_OFA6Bar.fb_6BarOFA_Alarm._AbortStateTimer
    Label (459,789 134x30), "Abort Running Timer"
    Label (723,793 49x30), "Sec"
    Textfield (208,691 123x30), "%d", text variable: fbDebugColumn.fb_facility_DewPoint_OFA6Bar.fb_DewPoint_Alarm._WarningStateTimer
    Label (72,692 134x30), "Warning Running Timer"
    Label (336,696 49x30), "Sec"
    Textfield (207,743 123x30), "%d", text variable: fbDebugColumn.fb_facility_DewPoint_OFA6Bar.fb_DewPoint_Alarm._AlarmStateTimer
    Label (71,744 134x30), "Alarm Running Timer"
    Label (335,748 49x30), "Sec"
    Textfield (209,794 123x30), "%d", text variable: fbDebugColumn.fb_facility_DewPoint_OFA6Bar.fb_DewPoint_Alarm._AbortStateTimer
    Label (73,795 134x30), "Abort Running Timer"
    Label (337,799 49x30), "Sec"
    Line (411,874) (416,104)
END_VISUALIZATION

// ---- VISUs/HMI_ManualCommand.TcVIS
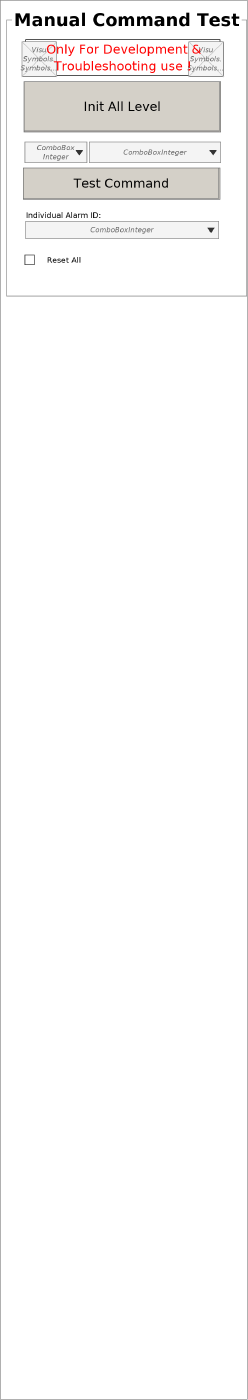
VISUALIZATION HMI_ManualCommand  // 354x1995
    GroupBox (9,20 343x402), "Manual Command Test"
        ComboBoxInteger (26,182 89x30), variable: iHMICbLevelSelection, text list: 'LevelTxtList'
    Button (33,239 281x45), "Test Command"
        tap TestManually.bTestCommand
    ComboBoxInteger (36,315 276x25), variable: TestManually.iAlarmCode, text list: 'AlarmTxtList'
    Checkbox (33,355 37x30), variable: bHMIResetAllAlarm
    Label (64,356 183x30), "Reset All"
    Label (34,292 215x30), "Individual Alarm ID:"
    Rectangle (9,1159 296x834), invisible if: bEnableManualCommandTest1 AND bEnableManualCommandTest2
    ComboBoxInteger (127,202 188x30), variable: iHMICbCmdSelection, text list: 'CmdTxtList'
    Button (34,116 281x72), "Init All Level"
        tap TestManually.bInitialiseAll
    Rectangle (36,56 278x52)
    Image (31,59 50x50), image: VisuSymbols.Symbols.Caution
    Image (269,59 50x50), image: VisuSymbols.Symbols.Caution
    Label (63,56 221x29), "Only For Development &"
    Label (74,80 210x29), "Troubleshooting use !"
END_VISUALIZATION

// ---- VISUs/HMI_OFA_Monitor.TcVIS
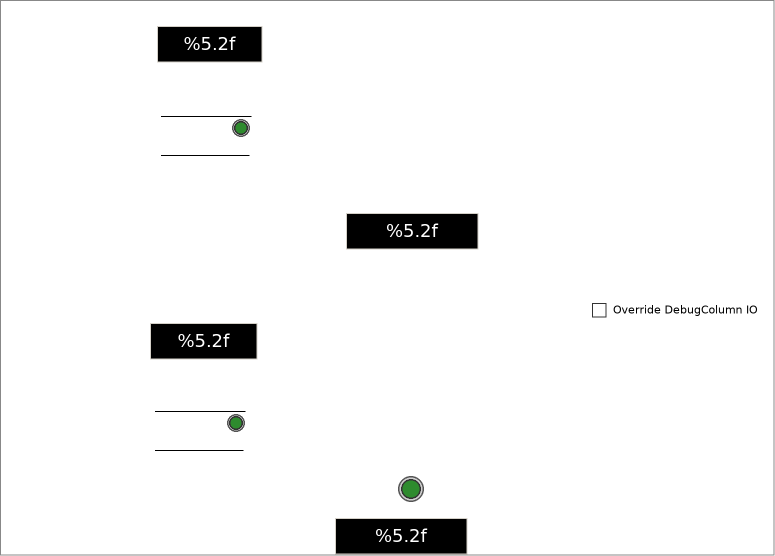
VISUALIZATION HMI_OFA_Monitor  // 775x556, background image ImageCollection.OFA Flow
    Lamp1 (396,474 30x30), variable: stDebugStation.fbDBStnSeq.stDebugStationDIO.opDBStnBypassAPAirSupplySol, style: Lamp-Lamp1-Green
    Textfield (157,26 105x36), "%5.2f", text variable: fbDebugColumn.stDebugColumnDIO.ipDBColumnTstAirPressure, input disabled if: TRUE
    Textfield (150,323 107x36), "%5.2f", text variable: fbDebugColumn.stDebugColumnDIO.ipDBColumnAPAirPressure, input disabled if: TRUE
    Rectangle (296,39 439x145)
    Rectangle (289,335 439x120)
    Lamp1 (226,413 20x20), variable: fbDebugColumn.stDebugColumnDIO.opDBColumnAPAirSol, style: Lamp-Lamp1-Green
    Lamp1 (231,118 20x20), variable: fbDebugColumn.stDebugColumnDIO.opDBColumnTstAirSol, style: Lamp-Lamp1-Green
    Textfield (346,213 132x36), "%5.2f", text variable: stDebugStation.fbDBStnSeq.stDebugStationDIO.ipDBStnTstAirLeakFlowSensor, input disabled if: TRUE
    Textfield (335,518 132x36), "%5.2f", text variable: stDebugStation.fbDBStnSeq.stDebugStationDIO.ipDBStnAPAirLeakFlowSensor, input disabled if: TRUE
    Line (155,411) (245,411)
    Line (155,450) (243,450)
    Line (161,116) (251,116)
    Line (161,155) (249,155)
    Checkbox (590,295 183x30), "Override DebugColumn IO"
END_VISUALIZATION

// ---- VISUs/HMI_PCWBehaviour.TcVIS
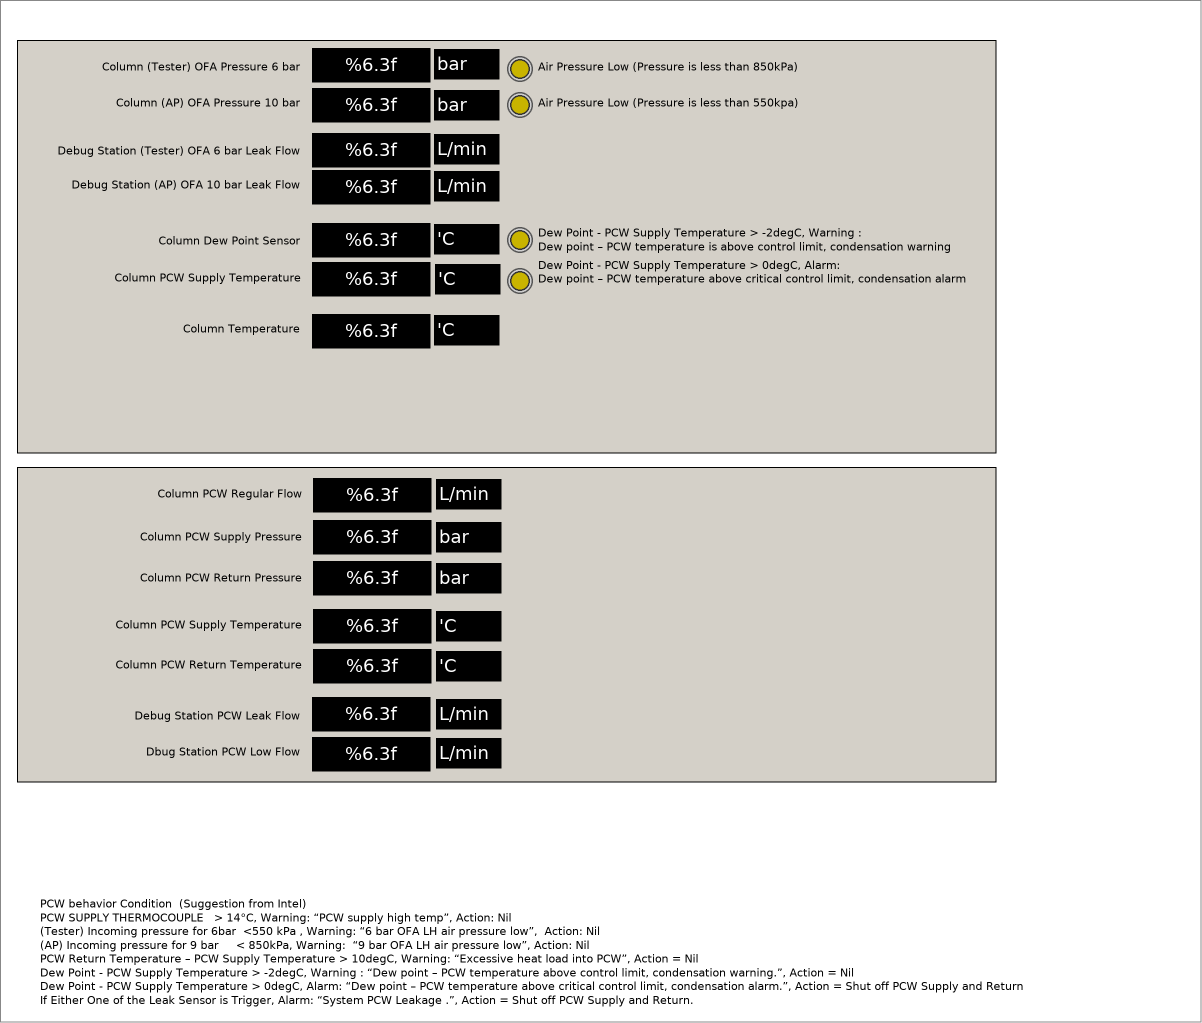
VISUALIZATION HMI_PCWBehaviour  // 1202x1023
    Rectangle (17,467 979x315)
    Rectangle (17,40 979x413)
    Textfield (311,47 120x36), "%6.3f", text variable: fbDebugColumn.stDebugColumnDIO.ipDBColumnTstAirPressure, input disabled if: TRUE
    Textfield (311,87 120x36), "%6.3f", text variable: fbDebugColumn.stDebugColumnDIO.ipDBColumnAPAirPressure, input disabled if: TRUE
    Textfield (311,132 120x36), "%6.3f", text variable: stDebugStation.fbDBStnSeq.stDebugStationDIO.ipDBStnTstAirLeakFlowSensor, input disabled if: TRUE
    Textfield (311,169 120x36), "%6.3f", text variable: stDebugStation.fbDBStnSeq.stDebugStationDIO.ipDBStnAPAirLeakFlowSensor, input disabled if: TRUE
    Label (42,136 261x30), "Debug Station (Tester) OFA 6 bar Leak Flow"
    Label (35,170 268x30), "Debug Station (AP) OFA 10 bar Leak Flow"
    Label (51,52 252x30), "Column (Tester) OFA Pressure 6 bar"
    Label (72,88 231x30), "Column (AP) OFA Pressure 10 bar"
    Textfield (311,696 120x36), "%6.3f", text variable: stDebugStation.fbDBStnSeq.stDebugStationDIO.ipDBStnPCWLeakFlowSensor, input disabled if: TRUE
    Textfield (311,736 120x36), "%6.3f", text variable: stDebugStation.fbDBStnSeq.stDebugStationDIO.ipDBStnPCWLowFlowSensor, input disabled if: TRUE
    Label (101,701 202x30), "Debug Station PCW Leak Flow"
    Label (55,737 248x30), "Dbug Station PCW Low Flow"
    Textfield (312,648 120x36), "%6.3f", text variable: fbDebugColumn.stDebugColumnDIO.ipDBColumnPCWReturnTemperature, input disabled if: TRUE
    Textfield (312,560 120x36), "%6.3f", text variable: fbDebugColumn.stDebugColumnDIO.ipDBColumnPCWReturnPressure, input disabled if: TRUE
    Textfield (312,477 120x36), "%6.3f", text variable: fbDebugColumn.stDebugColumnDIO.ipDBColumnPCWRegularFlowSensor, input disabled if: TRUE
    Textfield (312,519 120x36), "%6.3f", text variable: fbDebugColumn.stDebugColumnDIO.ipDBColumnPCWSupplyPressure, input disabled if: TRUE
    Textfield (312,608 120x36), "%6.3f", text variable: fbDebugColumn.stDebugColumnDIO.ipDBColumnPCWSupplyTemperature, input disabled if: TRUE
    Label (94,479 211x30), "Column PCW Regular Flow"
    Label (97,522 208x30), "Column PCW Supply Pressure"
    Label (122,563 183x30), "Column PCW Return Pressure"
    Label (76,610 229x30), "Column PCW Supply Temperature"
    Label (92,650 213x30), "Column PCW Return Temperature"
    Rectangle (436,479 65x30), "L/min"
    Rectangle (436,522 65x30), "bar"
    Rectangle (436,563 65x30), "bar"
    Rectangle (436,611 65x30), "'C"
    Rectangle (436,651 65x30), "'C"
    Rectangle (436,699 65x30), "L/min"
    Rectangle (436,738 65x30), "L/min"
    Rectangle (434,49 65x30), "bar"
    Rectangle (434,90 65x30), "bar"
    Rectangle (434,134 65x30), "L/min"
    Rectangle (434,171 65x30), "L/min"
    Textfield (311,222 120x36), "%6.3f", text variable: stDebugStation.fbDBStnSeq.stDebugStationDIO.ipDBStnTstAirLeakFlowSensor, input disabled if: TRUE
    Textfield (311,313 120x36), "%6.3f", text variable: fbDebugColumn.stDebugColumnDIO.ipDBColumnTempSensor, input disabled if: TRUE
    Label (124,226 179x30), "Column Dew Point Sensor"
    Label (153,314 150x30), "Column Temperature"
    Rectangle (434,224 65x30), "'C"
    Rectangle (434,315 65x30), "'C"
    Label (30,897 1170x124), "PCW behavior Condition (Suggestion from Intel) PCW SUPPLY THERMOCOUPLE > 14°C, Warning: “PCW supply high temp”, Action: Nil (Tester) Incoming pressure for 6bar <550 kPa , Warning: “6 bar OFA LH air pressure low”, Action: Nil (AP) Incoming pressure for 9 bar < 850kPa, Warning: “9 bar OFA LH air pressure low”, Action: Nil PCW Return Temperature – PCW Supply Temperature > 10degC, Warning: “Excessive heat load into PCW”, Action = Nil Dew Point - PCW Supply Temperature > -2degC, Warning : “Dew point – PCW temperature above control limit, condensation warning.”, Action = Nil Dew Point - PCW Supply Temperature > 0degC, Alarm: “Dew point – PCW temperature above critical control limit, condensation alarm.”, Action = Shut off PCW Supply and Return If Either One of the Leak Sensor is Trigger, Alarm: “System PCW Leakage .”, Action = Shut off PCW Supply and Return."
    Lamp1 (505,90 30x30), style: Lamp-Lamp1-Yellow
    Label (535,88 376x30), "Air Pressure Low (Pressure is less than 550kpa)"
    Lamp1 (505,54 30x30), style: Lamp-Lamp1-Yellow
    Label (535,52 376x30), "Air Pressure Low (Pressure is less than 850kPa)"
    Textfield (311,261 120x36), "%6.3f", text variable: fbDebugColumn.stDebugColumnDIO.ipDBColumnPCWSupplyTemperature, input disabled if: TRUE
    Label (75,263 229x30), "Column PCW Supply Temperature"
    Rectangle (435,264 65x30), "'C"
    Lamp1 (505,266 30x30), style: Lamp-Lamp1-Yellow
    Label (535,264 436x30), "Dew Point - PCW Supply Temperature > 0degC, Alarm: Dew point – PCW temperature above critical control limit, condensation alarm"
    Lamp1 (505,225 30x30), style: Lamp-Lamp1-Yellow
    Label (535,225 436x27), "Dew Point - PCW Supply Temperature > -2degC, Warning : Dew point – PCW temperature is above control limit, condensation warning"
END_VISUALIZATION

// ---- VISUs/HMI_PCW_Monitor.TcVIS
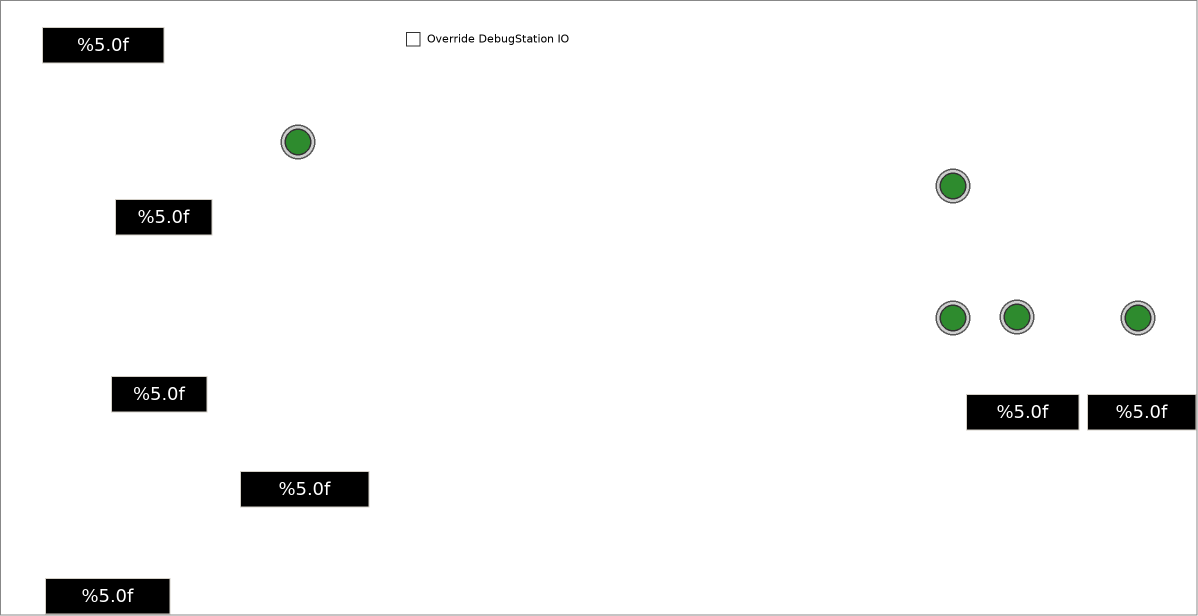
VISUALIZATION HMI_PCW_Monitor  // 1198x616, background image ImageCollection.PCW Flow
    Lamp1 (997,297 40x40), variable: stDebugStation.fbDBStnSeq.stDebugStationDIO.opDBStnLeakFlowPCWValve, style: Lamp-Lamp1-Green
    Textfield (966,394 113x36), "%5.0f", text variable: stDebugStation.fbDBStnSeq.stDebugStationDIO.ipDBStnPCWLeakFlowSensor, input disabled if: TRUE
    Textfield (1087,394 109x36), "%5.0f", text variable: stDebugStation.fbDBStnSeq.stDebugStationDIO.ipDBStnPCWLowFlowSensor, input disabled if: TRUE
    Lamp1 (1118,298 40x40), variable: stDebugStation.fbDBStnSeq.stDebugStationDIO.opDBStnLowFlowPCWValve, style: Lamp-Lamp1-Green
    Lamp1 (933,298 40x40), variable: stDebugStation.fbDBStnSeq.stDebugStationDIO.opDBStnPCWFlowBypassValve, style: Lamp-Lamp1-Green
    Lamp1 (933,166 40x40), variable: stDebugStation.fbDBStnSeq.stDebugStationDIO.opDBStnPCWValve, style: Lamp-Lamp1-Green
    Lamp1 (278,122 40x40), variable: fbDebugColumn.stDebugColumnDIO.opDBColumnPCWValve, style: Lamp-Lamp1-Green
    Textfield (111,376 96x36), "%5.0f", text variable: fbDebugColumn.stDebugColumnDIO.ipDBColumnPCWReturnTemperature, input disabled if: TRUE
    Textfield (45,578 125x36), "%5.0f", text variable: fbDebugColumn.stDebugColumnDIO.ipDBColumnPCWReturnPressure, input disabled if: TRUE
    Textfield (240,471 129x36), "%5.0f", text variable: fbDebugColumn.stDebugColumnDIO.ipDBColumnPCWRegularFlowSensor, input disabled if: TRUE
    Textfield (42,27 122x36), "%5.0f", text variable: fbDebugColumn.stDebugColumnDIO.ipDBColumnPCWSupplyPressure, input disabled if: TRUE
    Textfield (115,199 97x36), "%5.0f", text variable: fbDebugColumn.stDebugColumnDIO.ipDBColumnPCWSupplyTemperature, input disabled if: TRUE
    Rectangle (410,154 428x305)
    Rectangle (468,145 63x323)
    Rectangle (689,144 63x324)
    Rectangle (586,144 63x323)
    Checkbox (404,24 183x30), "Override DebugStation IO"
END_VISUALIZATION

